# B&R Automation Studio project Embraco_LinkaNaOdlievanieRotorov_DokoncovaciaStanica_Rev2 (part 3)

#### Main.st - Init, cyclic, exit code
```iecst
PROGRAM _INIT
	(* Insert code here *)

END_PROGRAM

PROGRAM _CYCLIC

	//Volanie podprogramov//
	OvladanieGripra;
	OvladaniePojazdu;
	OvladanieZdvihu;

	//Volanie funkcie SequenceControl//
	SequenceControl(SC:= SC_VstupnyManipulator);

	//Reset sekcie //
	IF VstupManipulator_Reset OR NOT BezpOkruhOplotenia_Aktivovany OR PoruchaVstupManipulator THEN
		SC_VstupnyManipulator.Step:= 0;
	END_IF

	CASE SC_VstupnyManipulator.Step OF

		0:
			SC_VstupnyManipulator.StepName:='0 - Nulovanie';
			SC_OvlGripra.Step:= 0;
			SC_OvlServoPojazdu.Step:= 0;
			SC_OvlZdvihu.Step:= 0;
			VstupManipulator_Automat:= FALSE;
			VstupManipulator_KoniecVyroby:= FALSE;
			VstupManipulator_KoniecCyklu:= FALSE;
			VstupManipulator_Manual:= FALSE;
			VstupManipulator_PoINIT:= FALSE;
			VstupManipulator_Reset:= FALSE;
			VstupManipulator_PojazdVPOZICI:= FALSE;
			VstupManipulator_UkoncilCyklus:= FALSE;
			Zariadenie_PAUZA:= FALSE;
			VstupManipulator_OdobralRotor:= FALSE;
			IF BezpOkruhOplotenia_Aktivovany AND NOT PoruchaVstupManipulator THEN
				SC_VstupnyManipulator.ResetStep:= TRUE;
				SC_VstupnyManipulator.Step:= 1;
			END_IF

		1:
			SC_VstupnyManipulator.StepName:='1 - Rozhodnutie o cinnosti';
			IF VstupManipulator_Automat THEN
				SC_VstupnyManipulator.Step:= 2;
			ELSIF VstupManipulator_Manual THEN
				SC_VstupnyManipulator.Step:= 700;
			END_IF

		//********************************************************Inicializácia****************************************************************************//

		2:
			SC_VstupnyManipulator.StepName:='2 - Inicializacia - cakanie na spustenie';
			SC_VstupnyManipulator.IdleTime.PT:= T#500ms;
			SC_VstupnyManipulator.AlarmTime.PT:= T#5s;
			SC_VstupnyManipulator.IdleTime.IN:= TRUE;

			IF SC_VstupnyManipulator.IdleTime.Q THEN
				SC_VstupnyManipulator.ResetStep:= TRUE;
				SC_VstupnyManipulator.Step:= 3;
			END_IF

		3:
			SC_VstupnyManipulator.StepName:='3 - Inicializacia - kontrola home serva';
			SC_VstupnyManipulator.IdleTime.PT:= T#500ms;
			SC_VstupnyManipulator.AlarmTime.PT:= T#5s;

			IF Motion[1].status.DriveStatus.HomingOk THEN
				SC_VstupnyManipulator.ResetStep:= TRUE;
				SC_VstupnyManipulator.Step:= 5;
			ELSE
				SC_VstupnyManipulator.ResetStep:= TRUE;
				SC_VstupnyManipulator.Step:= 4;
			END_IF

		4:
			SC_VstupnyManipulator.StepName:='4 - Inicializacia - homing serva';
			SC_VstupnyManipulator.IdleTime.PT:= T#1s;
			SC_VstupnyManipulator.AlarmTime.PT:= T#5s;

			IF NOT SC_VstupnyManipulator.Switch1 THEN
				VstupManipulator_PojazdHOME:= TRUE;
				SC_VstupnyManipulator.Switch1:= TRUE;
			END_IF

			IF Motion[1].status.DriveStatus.HomingOk THEN
				SC_VstupnyManipulator.IdleTime.IN:= TRUE;
			END_IF

			IF Motion[1].status.DriveStatus.HomingOk AND SC_VstupnyManipulator.IdleTime.Q AND Motion[1].state.StandStill THEN
				SC_VstupnyManipulator.ResetStep:= TRUE;
				SC_VstupnyManipulator.Step:= 6;
			END_IF

		5:
			SC_VstupnyManipulator.StepName:='5 - Inicializacia - zodvihnutie gripra';
			SC_VstupnyManipulator.IdleTime.PT:= T#500ms;
			SC_VstupnyManipulator.AlarmTime.PT:= T#5s;

			IF NOT SC_VstupnyManipulator.Switch1 THEN
				Zdvih_Manipulatora:= TRUE;
				SC_VstupnyManipulator.Switch1:= TRUE;
			END_IF

			IF diVstupManipul_ZasunutyHore THEN
				SC_VstupnyManipulator.ResetStep:= TRUE;
				SC_VstupnyManipulator.Step:= 6;
			END_IF

		6:
			SC_VstupnyManipulator.StepName:='6 - Inicializacia - rozhodnutie o presunu manipulatora';
			SC_VstupnyManipulator.IdleTime.PT:= T#200ms;
			SC_VstupnyManipulator.AlarmTime.PT:= T#5s;

			IF diVstupManipul_GriperOtvoreny AND diVstupManipul_GriperZatvoreny THEN
				Alarmy[21]:= TRUE;
				PoruchaVstupManipulator:= TRUE;
			ELSIF diVstupManipul_GriperOtvoreny AND NOT diVstupManipul_GriperZatvoreny THEN
				VstupManipulator_PoINIT:= TRUE;
				SC_VstupnyManipulator.ResetStep:= TRUE;
				SC_VstupnyManipulator.Step:= 125;
			ELSIF NOT diVstupManipul_GriperOtvoreny AND diVstupManipul_GriperZatvoreny THEN
				VstupManipulator_PoINIT:= TRUE;
				SC_VstupnyManipulator.ResetStep:= TRUE;
				SC_VstupnyManipulator.Step:= 110;
			END_IF

		//********************************************************Automatický režim****************************************************************************//
		100:
			SC_VstupnyManipulator.StepName:='100 - Automaticky rezim - cakanie na odobratie rotora';
			SC_VstupnyManipulator.IdleTime.PT:= T#3s;
			SC_VstupnyManipulator.AlarmTime.PT:= T#5s;
			SC_VstupnyManipulator.IdleTime.IN:= TRUE;

			IF VstupManipulator_KoniecCyklu THEN
				SC_VstupnyManipulator.ResetStep:= TRUE;
				SC_VstupnyManipulator.Step:= 0;
			ELSIF diVstupManipul_GriperOtvoreny AND NOT diVstupManipul_GriperZatvoreny AND diVstupDopr_PritomnostRotora AND diVstupDopr_ZdvihRotora_HORE AND NOT VstupManipulator_KoniecVyroby THEN
				SC_VstupnyManipulator.ResetStep:= TRUE;
				SC_VstupnyManipulator.Step:= 101;
			ELSIF diVstupManipul_GriperZatvoreny AND NOT diVstupManipul_GriperOtvoreny THEN
				SC_VstupnyManipulator.ResetStep:= TRUE;
				SC_VstupnyManipulator.Step:= 108;
			ELSIF SC_VstupnyManipulator.IdleTime.Q AND Stol_Automat THEN
				VstupManipulator_UkoncilCyklus:= TRUE;
				SC_VstupnyManipulator.ResetStep:= TRUE;
				SC_VstupnyManipulator.Step:= 132;
			ELSIF VstupManipulator_KoniecVyroby AND NOT Stol_Automat THEN
				SC_VstupnyManipulator.ResetStep:= TRUE;
				SC_VstupnyManipulator.Step:= 0;
			END_IF

		101:
			SC_VstupnyManipulator.StepName:='101 - Automaticky rezim - zostup manipulatora nad vstupny dopravnik';
			SC_VstupnyManipulator.IdleTime.PT:= T#1s;
			SC_VstupnyManipulator.AlarmTime.PT:= T#5s;
			SC_VstupnyManipulator.IdleTime.IN:= TRUE;

			IF NOT SC_VstupnyManipulator.Switch1 THEN
				Zostup_Manipulatora:= TRUE;
				SC_VstupnyManipulator.Switch1:= TRUE;
			END_IF

			IF diVstupManipul_VysunutyDole THEN
				SC_VstupnyManipulator.ResetStep:= TRUE;
				SC_VstupnyManipulator.Step:= 102;
			END_IF

		102:
			SC_VstupnyManipulator.StepName:='102 - Automaticky rezim - zatvorenie gripra manipulatora';
			SC_VstupnyManipulator.IdleTime.PT:= T#500ms;
			SC_VstupnyManipulator.AlarmTime.PT:= T#5s;

			IF NOT SC_VstupnyManipulator.Switch1 THEN
				Zatvor_Griper:= TRUE;
				SC_VstupnyManipulator.Switch1:= TRUE;
			END_IF

			IF diVstupManipul_GriperZatvoreny THEN
				SC_VstupnyManipulator.ResetStep:= TRUE;
				SC_VstupnyManipulator.Step:= 103;
			END_IF

		103:
			SC_VstupnyManipulator.StepName:='103 - Automaticky rezim - otvorenie gripra manipulatora';
			SC_VstupnyManipulator.IdleTime.PT:= T#500ms;
			SC_VstupnyManipulator.AlarmTime.PT:= T#5s;

			IF NOT SC_VstupnyManipulator.Switch1 AND SC_OvlGripra.Step = 1 THEN
				Otvor_Griper:= TRUE;
				SC_VstupnyManipulator.Switch1:= TRUE;
			END_IF

			IF diVstupManipul_GriperOtvoreny THEN
				SC_VstupnyManipulator.ResetStep:= TRUE;
				SC_VstupnyManipulator.Step:= 104;
			END_IF

		104:
			SC_VstupnyManipulator.StepName:='104 - Automaticky rezim - zatvorenie gripra manipulatora';
			SC_VstupnyManipulator.IdleTime.PT:= T#500ms;
			SC_VstupnyManipulator.AlarmTime.PT:= T#5s;

			IF NOT SC_VstupnyManipulator.Switch1 AND SC_OvlGripra.Step = 1 THEN
				Zatvor_Griper:= TRUE;
				SC_VstupnyManipulator.Switch1:= TRUE;
			END_IF

			IF diVstupManipul_GriperZatvoreny THEN
				SC_VstupnyManipulator.ResetStep:= TRUE;
				SC_VstupnyManipulator.Step:= 108;
			END_IF

		108:
			SC_VstupnyManipulator.StepName:='102 - Automaticky rezim - zdvih manipulatora nad vstupny dopravnik, zistovanie NG kusu';
			SC_VstupnyManipulator.IdleTime.PT:= T#500ms;
			SC_VstupnyManipulator.AlarmTime.PT:= T#5s;
			SC_VstupnyManipulator.IdleTime.IN:= TRUE;

			IF NOT SC_VstupnyManipulator.Switch1 THEN
				Zdvih_Manipulatora:= TRUE;
				SC_VstupnyManipulator.Switch1:= TRUE;
			END_IF

			IF EDGEPOS(diVstupManipul_SpodSnimacNG_Kusu = TRUE) THEN
				IF diVstupManipul_HornSnimacNG_Kusu THEN
					VstupManipulator_Drzi_NG_Kus:= FALSE;
				ELSIF Zariadenie_PrebiehaRevorkRezim THEN
					VstupManipulator_Drzi_NG_Kus:= FALSE;
				ELSE
					VstupManipulator_Drzi_NG_Kus:= TRUE;
				END_IF
			END_IF

			IF diVstupManipul_ZasunutyHore THEN
				SC_VstupnyManipulator.ResetStep:= TRUE;
				SC_VstupnyManipulator.Step:= 110;
			END_IF

		110:
			SC_VstupnyManipulator.StepName:='104 - Automaticky rezim - presun manipulatora na poziciu vkladania';
			SC_VstupnyManipulator.IdleTime.PT:= T#500ms;
			SC_VstupnyManipulator.AlarmTime.PT:= T#5s;

			VstupManipulator_ZadanaPozMM:= TP_VstupManip_PoziciaUkladania; //9 mm

			IF NOT SC_VstupnyManipulator.Switch1 AND SC_OvlServoPojazdu.Step = 1 THEN
				ServoPojazd_Polohuj:= TRUE;
				SC_VstupnyManipulator.Switch1:= TRUE;
			END_IF

			IF VstupManipulator_PojazdVPOZICI AND (VstupManipulator_AktualPozMM = TP_VstupManip_PoziciaUkladania) THEN
				VstupManipulator_PojazdVPOZICI:= FALSE;
				SC_VstupnyManipulator.ResetStep:= TRUE;
				SC_VstupnyManipulator.Step:= 120;
			END_IF

		120:
			SC_VstupnyManipulator.StepName:='120 - Automaticky rezim - kontrola stola';
			SC_VstupnyManipulator.IdleTime.PT:= T#500ms;
			SC_VstupnyManipulator.AlarmTime.PT:= T#5s;

			IF Stol_PoINIT AND NOT VstupManipulator_UkoncilCyklus AND diStol_SnimacPolohyStola AND NOT diStol_PritomnostRotoraVstup THEN
				SC_VstupnyManipulator.ResetStep:= TRUE;
				SC_VstupnyManipulator.Step:= 122;
			ELSIF Stol_PoINIT AND NOT VstupManipulator_UkoncilCyklus AND diStol_SnimacPolohyStola AND diStol_PritomnostRotoraVstup THEN
				VstupManipulator_UkoncilCyklus:= TRUE;
				SC_VstupnyManipulator.ResetStep:= TRUE;
				SC_VstupnyManipulator.Step:= 132;
			ELSIF VstupManipulator_KoniecCyklu THEN
				SC_VstupnyManipulator.ResetStep:= TRUE;
				SC_VstupnyManipulator.Step:= 0;
			END_IF

		122:
			SC_VstupnyManipulator.StepName:='122 - Automaticky rezim - polozenie rotora na stol';
			SC_VstupnyManipulator.IdleTime.PT:= T#200ms;
			SC_VstupnyManipulator.AlarmTime.PT:= T#5s;
			SC_VstupnyManipulator.AlarmTime.IN:= TRUE;

			IF NOT SC_VstupnyManipulator.Switch1 AND diStol_SnimacPolohyStola AND NOT diStol_PritomnostRotoraVstup AND Stol.IN.CentrovanieVysunute=1 THEN
				Zostup_Manipulatora:= TRUE;
				SC_VstupnyManipulator.Switch1:= TRUE;
			END_IF

			IF diVstupManipul_ZdvihStredPoloha THEN
				SC_VstupnyManipulator.IdleTime.IN:= TRUE;
			END_IF

			IF diVstupManipul_VysunutyDole OR SC_VstupnyManipulator.IdleTime.Q THEN
				SC_VstupnyManipulator.ResetStep:= TRUE;
				SC_VstupnyManipulator.Step:= 123;
			END_IF

			IF SC_VstupnyManipulator.AlarmTime.Q THEN
				Alarmy[23]:= TRUE;
				PoruchaVstupManipulator:= TRUE;
			END_IF

		123:
			SC_VstupnyManipulator.StepName:='123 - Automaticky rezim - otvorenie gripra manipulatora';
			SC_VstupnyManipulator.IdleTime.PT:= T#500ms;
			SC_VstupnyManipulator.AlarmTime.PT:= T#5s;

			IF NOT SC_VstupnyManipulator.Switch1 THEN
				Otvor_Griper:= TRUE;
				SC_VstupnyManipulator.Switch1:= TRUE;
			END_IF

			IF diVstupManipul_GriperOtvoreny AND diVstupManipul_VysunutyDole THEN
				IF VstupManipulator_Drzi_NG_Kus THEN
					Stol_NG_KusNaStole:= TRUE;
				ELSE
					Stol_NG_KusNaStole:= FALSE;
				END_IF
				VstupManipulator_Drzi_NG_Kus:= FALSE;
				SC_VstupnyManipulator.ResetStep:= TRUE;
				SC_VstupnyManipulator.Step:= 124;
			END_IF

		124:
			SC_VstupnyManipulator.StepName:='124 - Automaticky rezim - zdvih manipulatora nad stol, vystavenie signalu ukoncenie cyklu';
			SC_VstupnyManipulator.IdleTime.PT:= T#500ms;
			SC_VstupnyManipulator.AlarmTime.PT:= T#5s;

			IF NOT SC_VstupnyManipulator.Switch1 AND SC_OvlZdvihu.Step = 1 THEN
				Zdvih_Manipulatora:= TRUE;
				Stol.OUT.CentrovanieVysunut:=0;
				Stol.OUT.CentrovanieZasunut:=1;
				SC_VstupnyManipulator.Switch1:= TRUE;
			END_IF

			IF diVstupManipul_ZasunutyHore AND Stol.IN.CentrovanieZasunute=1 THEN
				IF diStol_PritomnostRotoraVstup THEN
					VstupManipulator_UkoncilCyklus:= TRUE;
				END_IF
				SC_VstupnyManipulator.ResetStep:= TRUE;
				SC_VstupnyManipulator.Step:= 125;
			END_IF

		125:
			SC_VstupnyManipulator.StepName:='125 - Automaticky rezim - presun manipulatora na poziciu odoberania';
			SC_VstupnyManipulator.IdleTime.PT:= T#500ms;
			SC_VstupnyManipulator.AlarmTime.PT:= T#5s;

			VstupManipulator_ZadanaPozMM:= TP_VstupManip_PoziciaOdoberania;//602.0;

			IF NOT SC_VstupnyManipulator.Switch1 AND SC_OvlServoPojazdu.Step = 1 THEN
				ServoPojazd_Polohuj:= TRUE;
				SC_VstupnyManipulator.Switch1:= TRUE;
			END_IF

			IF VstupManipulator_PojazdVPOZICI AND (VstupManipulator_AktualPozMM = TP_VstupManip_PoziciaOdoberania) THEN
				VstupManipulator_PojazdVPOZICI:= FALSE;
				SC_VstupnyManipulator.ResetStep:= TRUE;
				SC_VstupnyManipulator.Step:= 100;
			END_IF

		132:
			SC_VstupnyManipulator.StepName:='132 - Automaticky rezim - cakanie na otocenie stola';
			SC_VstupnyManipulator.IdleTime.PT:= T#500ms;
			SC_VstupnyManipulator.AlarmTime.PT:= T#5s;

			IF NOT VstupManipulator_UkoncilCyklus THEN
				SC_VstupnyManipulator.ResetStep:= TRUE;
				SC_VstupnyManipulator.Step:= 100;
			ELSIF VstupManipulator_KoniecVyroby AND NOT Stol_Automat THEN
				SC_VstupnyManipulator.ResetStep:= TRUE;
				SC_VstupnyManipulator.Step:= 0;
			ELSIF VstupManipulator_KoniecCyklu THEN
				SC_VstupnyManipulator.ResetStep:= TRUE;
				SC_VstupnyManipulator.Step:= 0;
			END_IF

		//********************************************************Ručný režim***********************************************************************************//
		700:
			SC_VstupnyManipulator.StepName:='700 - Rucny rezim';

			//Polohovanie manipulátora//
			IF RR_PoziciaOdoberania AND SC_OvlServoPojazdu.Step = 1 THEN
				VstupManipul_Rychlost_MM_s:= TP_VstupManip_RychlostPojazdu;
				VstupManipulator_ZadanaPozMM:= TP_VstupManip_PoziciaOdoberania;
				ServoPojazd_Polohuj:= TRUE;
			ELSIF RR_PoziciaVkladaniaStol AND SC_OvlServoPojazdu.Step = 1 THEN
				VstupManipul_Rychlost_MM_s:= TP_VstupManip_RychlostPojazdu;
				VstupManipulator_ZadanaPozMM:= TP_VstupManip_PoziciaUkladania;
				ServoPojazd_Polohuj:= TRUE;
			END_IF

	END_CASE

				END_PROGRAM

PROGRAM _EXIT
				(* Insert code here *)

				END_PROGRAM
```

#### Variables.var - Local variables
```iecst
VAR
	SC_OvlGripra : SequenceControlTyp;
	Otvor_Griper : BOOL;
	Zatvor_Griper : BOOL;
	SC_OvlZdvihu : SequenceControlTyp;
	Zdvih_Manipulatora : BOOL;
	Zostup_Manipulatora : BOOL;
	SC_OvlServoPojazdu : SequenceControlTyp;
	ServoPojazd_JoggVPRED : BOOL;
	ServoPojazd_JoggVZAD : BOOL;
	ServoPojazd_Polohuj : BOOL;
	KonstantaPojazd_MM : REAL;
	KonstantaPojazd_Servo : REAL;
	RR_PoziciaOdoberania : BOOL;
	RR_PoziciaVkladaniaStol : BOOL;
END_VAR
```

#### OvladanieGripra.st
```iecst
ACTION OvladanieGripra:

	//Volanie funkcie SequenceControl//
	SequenceControl(SC:= SC_OvlGripra);

	CASE SC_OvlGripra.Step OF

		0:
			SC_OvlGripra.StepName:= '0 - Nulovanie';
			Otvor_Griper:= FALSE;
			Zatvor_Griper:= FALSE;
			doVstupManipul_GriperOTVOR:= FALSE;
			doVstupManipul_GriperZATVOR:= FALSE;
			IF SC_VstupnyManipulator.Step <> 0 THEN
				SC_OvlGripra.ResetStep:= TRUE;
				SC_OvlGripra.Step:= 1;
			END_IF

		1:
			SC_OvlGripra.StepName:= '1 - Rozhodnutie o cinnosti';
			IF Otvor_Griper THEN
				SC_OvlGripra.Step:= 10;
			ELSIF Zatvor_Griper THEN
				SC_OvlGripra.Step:= 20;
			END_IF

		10:
			SC_OvlGripra.StepName:= '10 - Otvorenie gripra';
			SC_OvlGripra.IdleTime.PT:= T#3s;
			SC_OvlGripra.AlarmTime.PT:= T#3s;

			IF VstupManipulator_Manual THEN
				SC_OvlGripra.IdleTime.IN:= TRUE;
			ELSE
				SC_OvlGripra.AlarmTime.IN:= TRUE;
			END_IF

			IF NOT SC_OvlGripra.Switch1 THEN
				doVstupManipul_GriperOTVOR:= TRUE;
				SC_OvlGripra.Switch1:= TRUE;
			END_IF

			IF SC_OvlGripra.AlarmTime.Q THEN
				Alarmy[21]:= TRUE;
				PoruchaVstupManipulator:= TRUE;
			END_IF

			IF diVstupManipul_GriperOtvoreny OR SC_OvlGripra.IdleTime.Q THEN
				SC_OvlGripra.ResetStep:= TRUE;
				SC_OvlGripra.Step:= 0;
			END_IF

		20:
			SC_OvlGripra.StepName:= '20 - Zatvorenie gripra';
			SC_OvlGripra.IdleTime.PT:= T#3s;
			SC_OvlGripra.AlarmTime.PT:= T#3s;

			IF VstupManipulator_Manual THEN
				SC_OvlGripra.IdleTime.IN:= TRUE;
			ELSE
				SC_OvlGripra.AlarmTime.IN:= TRUE;
			END_IF

			IF NOT SC_OvlGripra.Switch1 THEN
				doVstupManipul_GriperZATVOR:= TRUE;
				SC_OvlGripra.Switch1:= TRUE;
			END_IF

			IF SC_OvlGripra.AlarmTime.Q THEN
				Alarmy[20]:= TRUE;
				PoruchaVstupManipulator:= TRUE;
			END_IF

			IF diVstupManipul_GriperZatvoreny OR SC_OvlGripra.IdleTime.Q THEN
				SC_OvlGripra.ResetStep:= TRUE;
				SC_OvlGripra.Step:= 0;
			END_IF

	END_CASE

END_ACTION
```

#### OvladanieZdvihu.st
```iecst
ACTION OvladanieZdvihu:

	//Volanie funkcie SequenceControl//
	SequenceControl(SC:= SC_OvlZdvihu);

	CASE SC_OvlZdvihu.Step OF

		0:
			SC_OvlZdvihu.StepName:= '0 - Nulovanie';
			Zdvih_Manipulatora:= FALSE;
			Zostup_Manipulatora:= FALSE;
			doVstupManipul_ZDVIH:= FALSE;
			doVstupManipul_ZOSTUP:= FALSE;
			IF SC_VstupnyManipulator.Step <> 0 THEN
				SC_OvlZdvihu.ResetStep:= TRUE;
				SC_OvlZdvihu.Step:= 1;
			END_IF

		1:
			SC_OvlZdvihu.StepName:= '1 - Rozhodnutie o cinnosti';
			IF Zdvih_Manipulatora THEN
				SC_OvlZdvihu.Step:= 10;
			ELSIF Zostup_Manipulatora THEN
				SC_OvlZdvihu.Step:= 20;
			END_IF

		10:
			SC_OvlZdvihu.StepName:= '10 - Zdvih manipulatora';
			SC_OvlZdvihu.IdleTime.PT:= T#3s;
			SC_OvlZdvihu.AlarmTime.PT:= T#3s;

			IF VstupManipulator_Manual THEN
				SC_OvlZdvihu.IdleTime.IN:= TRUE;
			ELSE
				SC_OvlZdvihu.AlarmTime.IN:= TRUE;
			END_IF

			IF NOT SC_OvlZdvihu.Switch1 THEN
				doVstupManipul_ZDVIH:= TRUE;
				SC_OvlZdvihu.Switch1:= TRUE;
			END_IF

			IF SC_OvlZdvihu.AlarmTime.Q THEN
				Alarmy[22]:= TRUE;
				PoruchaVstupManipulator:= TRUE;
			END_IF

			IF diVstupManipul_ZasunutyHore OR SC_OvlZdvihu.IdleTime.Q THEN
				SC_OvlZdvihu.ResetStep:= TRUE;
				SC_OvlZdvihu.Step:= 0;
			END_IF

		20:
			SC_OvlZdvihu.StepName:= '20 - Zostup manipulatora';
			SC_OvlZdvihu.IdleTime.PT:= T#2s;
			SC_OvlZdvihu.AlarmTime.PT:= T#3s;
			SC_OvlZdvihu.IdleTime.IN:= TRUE;

			IF VstupManipulator_Manual THEN
				SC_OvlZdvihu.IdleTime.IN:= TRUE;
			ELSE
				SC_OvlZdvihu.AlarmTime.IN:= TRUE;
			END_IF

			IF NOT SC_OvlZdvihu.Switch1 THEN
				doVstupManipul_ZOSTUP:= TRUE;
				SC_OvlZdvihu.Switch1:= TRUE;
			END_IF

			IF EDGEPOS (diVstupManipul_ZdvihStredPoloha = TRUE) THEN
				doVstupManipul_ZDVIH:= TRUE;
			END_IF

			IF SC_OvlZdvihu.AlarmTime.Q THEN
				Alarmy[23]:= TRUE;
				PoruchaVstupManipulator:= TRUE;
			END_IF

			IF diVstupManipul_VysunutyDole OR SC_OvlZdvihu.IdleTime.Q THEN
				SC_OvlZdvihu.ResetStep:= TRUE;
				SC_OvlZdvihu.Step:= 0;
			END_IF

	END_CASE

END_ACTION
```

#### OvladaniePojazdu.st
```iecst
ACTION OvladaniePojazdu:

	//Prepočet rýchlosti pojazdu manipulátora//
	KonstantaPojazd_MM:= 8;  //8mm
	KonstantaPojazd_Servo:= 800; //počet jednotiek za 8mm

	VstupManipul_Rychlost_MM_s:= TP_VstupManip_RychlostPojazdu;
	VstupManipulator_RychlostPolohov:= (VstupManipul_Rychlost_MM_s / KonstantaPojazd_MM) * KonstantaPojazd_Servo;
	VstupManipulator_RychlJoggingu:= (VstupManipul_RychlostJog_MM_s / KonstantaPojazd_MM) * KonstantaPojazd_Servo;
	VstupManipulator_AktualPozMM;

	//Volanie funkcie SequenceControl//
	SequenceControl(SC:= SC_OvlServoPojazdu);

	CASE SC_OvlServoPojazdu.Step OF

		0:
			SC_OvlServoPojazdu.StepName:= '0 - Nulovanie';
			ServoPojazd_JoggVPRED:= FALSE;
			ServoPojazd_JoggVZAD:= FALSE;
			ServoPojazd_Polohuj:= FALSE;
			VstupManipulator_PojazdHOME:= FALSE;
			Motion[1].cmd.home:= FALSE;
			Motion[1].cmd.moveAbsolute:= FALSE;
			Motion[1].cmd.moveJogNeg:= FALSE;
			Motion[1].cmd.moveJogPos:= FALSE;
			VstupManipulator_PrebiehaHoming:= FALSE;
			IF NOT SC_OvlServoPojazdu.Switch1 AND Motion[1].status.DriveStatus.HomingOk THEN
				Motion[1].cmd.halt:= TRUE;
				SC_OvlServoPojazdu.Switch1:= TRUE;
			END_IF
			IF SC_VstupnyManipulator.Step <> 0 THEN
				SC_OvlServoPojazdu.ResetStep:= TRUE;
				SC_OvlServoPojazdu.Step:= 1;
			END_IF

		1:
			SC_OvlServoPojazdu.StepName:= '1 - Rozhodnutie o cinnosti';
			IF ServoPojazd_JoggVPRED THEN
				SC_OvlServoPojazdu.Step:= 10;
			ELSIF ServoPojazd_JoggVZAD THEN
				SC_OvlServoPojazdu.Step:= 20;
			ELSIF ServoPojazd_Polohuj THEN
				SC_OvlServoPojazdu.Step:= 30;
			ELSIF VstupManipulator_PojazdHOME THEN
				SC_OvlServoPojazdu.Step:= 40;
			END_IF

		10:
			SC_OvlServoPojazdu.StepName:= '10 - Jogging VPRED';
			SC_OvlServoPojazdu.IdleTime.PT:= T#3s;
			SC_OvlServoPojazdu.AlarmTime.PT:= T#3s;

			Motion[1].par.velocityJog:= VstupManipulator_RychlJoggingu;
			Motion[1].par.acc := (VstupManipulator_RychlJoggingu*10);
			Motion[1].par.dec := (VstupManipulator_RychlJoggingu*10);

			IF NOT SC_OvlServoPojazdu.Switch1 THEN
				Motion[1].cmd.moveJogPos:= TRUE;
				SC_OvlServoPojazdu.Switch1:= TRUE;
			END_IF

			IF NOT ServoPojazd_JoggVPRED OR diVstupManipul_PrednyLimitSnimac OR VstupManipulator_AktualPozMM >= 610 OR NOT diVstupManipul_ZasunutyHore THEN
				SC_OvlServoPojazdu.ResetStep:= TRUE;
				SC_OvlServoPojazdu.Step:= 0;
			END_IF

		20:
			SC_OvlServoPojazdu.StepName:= '10 - Jogging VZAD';
			SC_OvlServoPojazdu.IdleTime.PT:= T#3s;
			SC_OvlServoPojazdu.AlarmTime.PT:= T#3s;

			Motion[1].par.velocityJog:= VstupManipulator_RychlJoggingu;
			Motion[1].par.acc := (VstupManipulator_RychlJoggingu*10);
			Motion[1].par.dec := (VstupManipulator_RychlJoggingu*10);

			IF NOT SC_OvlServoPojazdu.Switch1 THEN
				Motion[1].cmd.moveJogNeg:= TRUE;
				SC_OvlServoPojazdu.Switch1:= TRUE;
			END_IF

			IF NOT ServoPojazd_JoggVZAD OR diVstupManipul_ZadnyLimitSnimac OR VstupManipulator_AktualPozMM < 0 OR NOT diVstupManipul_ZasunutyHore THEN
				SC_OvlServoPojazdu.ResetStep:= TRUE;
				SC_OvlServoPojazdu.Step:= 0;
			END_IF

		30:
			SC_OvlServoPojazdu.StepName:= '30 - Start polohovanie pojazdu';
			SC_OvlServoPojazdu.IdleTime.PT:= T#100ms;
			SC_OvlServoPojazdu.AlarmTime.PT:= T#3s;
			SC_OvlServoPojazdu.IdleTime.IN:= TRUE;

			Motion[1].par.velocity:= VstupManipulator_RychlostPolohov;
			Motion[1].par.acc := (VstupManipulator_RychlostPolohov*10);
			Motion[1].par.dec := (VstupManipulator_RychlostPolohov*10);
			Motion[1].par.position:= (VstupManipulator_ZadanaPozMM * 100);

			IF NOT SC_OvlServoPojazdu.Switch1 AND SC_OvlServoPojazdu.IdleTime.Q THEN
				Motion[1].cmd.moveAbsolute:= TRUE;
				SC_OvlServoPojazdu.Switch1:= TRUE;
			END_IF

			IF NOT Motion[1].state.StandStill THEN
				SC_OvlServoPojazdu.ResetStep:= TRUE;
				SC_OvlServoPojazdu.Step:= 31;
			ELSIF (VstupManipulator_AktualPozMM = VstupManipulator_ZadanaPozMM) THEN
				SC_OvlServoPojazdu.ResetStep:= TRUE;
				SC_OvlServoPojazdu.Step:= 31;
			END_IF

		31:

			SC_OvlServoPojazdu.StepName:= '31 - Ukoncenie polohovanie pojazdu';
			SC_OvlServoPojazdu.IdleTime.PT:= T#3s;
			SC_OvlServoPojazdu.AlarmTime.PT:= T#3s;

			IF Motion[1].state.StandStill AND (VstupManipulator_AktualPozMM = VstupManipulator_ZadanaPozMM) THEN
				VstupManipulator_PojazdVPOZICI:= TRUE;
				SC_OvlServoPojazdu.ResetStep:= TRUE;
				SC_OvlServoPojazdu.Step:= 0;
			END_IF

			IF diVstupManipul_PrednyLimitSnimac OR diVstupManipul_ZadnyLimitSnimac THEN
				Alarmy[26]:= TRUE;
				PoruchaVstupManipulator:= TRUE;
			END_IF

		40:
			SC_OvlServoPojazdu.StepName:= '40 - Homing,zdvihnutie gripra';
			SC_OvlServoPojazdu.IdleTime.PT:= T#3s;
			SC_OvlServoPojazdu.AlarmTime.PT:= T#3s;

			IF NOT SC_OvlServoPojazdu.Switch1 THEN
				VstupManipulator_PrebiehaHoming:= TRUE;
				Zdvih_Manipulatora:= TRUE;
				SC_OvlServoPojazdu.Switch1:= TRUE;
			END_IF

			IF diVstupManipul_ZasunutyHore THEN
				SC_OvlServoPojazdu.ResetStep:= TRUE;
				SC_OvlServoPojazdu.Step:= 41;
			END_IF

		41:
			SC_OvlServoPojazdu.StepName:= '41 - Homing,spustenie';
			SC_OvlServoPojazdu.IdleTime.PT:= T#3s;
			SC_OvlServoPojazdu.AlarmTime.PT:= T#3s;

			IF NOT SC_OvlServoPojazdu.Switch1 THEN
				Motion[1].cmd.home:= TRUE;
				SC_OvlServoPojazdu.Switch1:= TRUE;
			END_IF

			IF Motion[1].state.Homing THEN
				SC_OvlServoPojazdu.ResetStep:= TRUE;
				SC_OvlServoPojazdu.Step:= 42;
			END_IF

		42:
			SC_OvlServoPojazdu.StepName:= '42 - Homing,ukoncenie';
			SC_OvlServoPojazdu.IdleTime.PT:= T#3s;
			SC_OvlServoPojazdu.AlarmTime.PT:= T#3s;

			IF Motion[1].status.DriveStatus.HomingOk AND Motion[1].state.StandStill THEN
				SC_OvlServoPojazdu.ResetStep:= TRUE;
				SC_OvlServoPojazdu.Step:= 0;
			END_IF

	END_CASE

END_ACTION
```

### Program Logical/Program/OtocnyStol (IEC)

#### Main.st - Init, cyclic, exit code
```iecst
PROGRAM _INIT
	(* Insert code here *)

END_PROGRAM

PROGRAM _CYCLIC

	//Volanie podprogramov//
    OvladanieOtacania;

    //Volanie funkcie SequenceControl//
    SequenceControl(SC:= SC_Stol);

    //Blokovanie otáčania stola//
    IF diMeranie_ZdvihSpodnaPoloha AND
        diRazenie_ZdvihSpodnaPoloha AND
        Vyrazanie.IN.VyrazanieJeDole AND
        diValcovanie_ZdvihSpodnaPoloha AND
        (diVstupManipul_ZasunutyHore OR VstupManipulator_AktualPozMM > 15) AND
        (diVystupManipul_ZasunutyHore OR VystupManipulator_AktualPozMM > 15) AND
        NOT diValcovanie_PritomnostNastroja AND
        diValc2_ZdvihRotoraZasunuty AND
        Vyrazanie.IN.CentrovanieOtvorene THEN
        Stol_BlokovanieOtacania:= FALSE;
    ELSE
        Stol_BlokovanieOtacania:= TRUE;
    END_IF

    //Reset sekcie //
    IF Stol_Reset OR NOT BezpOkruhOplotenia_Aktivovany OR PoruchaOtocnyStol THEN
        SC_Stol.Step:= 0;
    END_IF

    CASE SC_Stol.Step OF

        0:
            SC_Stol.StepName:='0 - Nulovanie';
            SC_OvlStola.Step:= 0;
            Stol_Automat:= FALSE;
            Stol_KoniecVyroby:= FALSE;
            Stol_KoniecCyklu:= FALSE;
            Stol_Manual:= FALSE;
            Stol_PoINIT:= FALSE;
            Stol_Reset:= FALSE;
            Stol_PrebehloOtocenie:= FALSE;
            Stol_CakaNaVstupnyManipulator:= FALSE;
            Stol_CakaNaStrihanie:= FALSE;
            Stol_CakaNaRazenie:= FALSE;
            Stol_CakaNaValcovanie:= FALSE;
            Stol_CakaNaMeranie:= FALSE;
            Stol_CakaNaVystupnyManipulator:= FALSE;
            //			Stol_Pozicia_1:= 0;
            //			Stol_Pozicia_2:= 0;
            //			Stol_Pozicia_3:= 0;
            PocetOtoceniStola:= 0;
            Stol_StavPrazdnyStol:= FALSE;
            CasTaktTime2.IN:= FALSE;
            CasTaktTime1.IN:= FALSE;
            TP_Stol_Centrovanie_VYSUN:= FALSE;
            TP_Stol_Centrovanie_ZASUN:= FALSE;
            IF BezpOkruhOplotenia_Aktivovany AND NOT PoruchaOtocnyStol THEN
                SC_Stol.ResetStep:= TRUE;
                SC_Stol.Step:= 1;
            END_IF

        1:
            SC_Stol.StepName:='1 - Rozhodnutie o cinnosti';
            IF Stol_Automat THEN
                CisloChyby:= 0;
                SC_Stol.Step:= 2;
            ELSIF Stol_Manual THEN
                SC_Stol.Step:= 700;
            END_IF

            //********************************************************Inicializácia****************************************************************************//

        2:
            SC_Stol.StepName:='2 - Inicializacia - cakanie na spustenie';
            SC_Stol.IdleTime.PT:= T#500ms;
            SC_Stol.AlarmTime.PT:= T#5s;
            SC_Stol.IdleTime.IN:= TRUE;

            IF SC_Stol.IdleTime.Q THEN
                SC_Stol.ResetStep:= TRUE;
                SC_Stol.Step:= 3;
            END_IF

        3:
            SC_Stol.StepName:='2 - Inicializacia - rozhodnutie o otoceni stola';
            SC_Stol.IdleTime.PT:= T#500ms;
            SC_Stol.AlarmTime.PT:= T#5s;

            IF diStol_SnimacPolohyStola THEN
                Stol.OUT.CentrovanieVysunut:=1;
                Stol.OUT.CentrovanieZasunut:=0;
                Stol_PoINIT:= TRUE;
                SC_Stol.ResetStep:= TRUE;
                IF Stol.IN.CentrovanieVysunute=1 THEN
                    SC_Stol.Step:= 100;
                END_IF
            ELSE
                SC_Stol.ResetStep:= TRUE;
                SC_Stol.Step:= 4;
            END_IF

        4:
            SC_Stol.StepName:='4 - Inicializacia - otocenie stola vpred';
            SC_Stol.IdleTime.PT:= T#500ms;
            SC_Stol.AlarmTime.PT:= T#5s;

            IF NOT SC_Stol.Switch1 AND NOT Stol_BlokovanieOtacania THEN
                Otacaj_VPRED:= TRUE;
                SC_Stol.Switch1:= TRUE;
            END_IF

            IF diStol_SnimacPolohyStola AND Stol_PrebehloOtocenie THEN
                Stol_PrebehloOtocenie:= FALSE;
                Stol_PoINIT:= TRUE;
                SC_Stol.ResetStep:= TRUE;
                SC_Stol.Step:= 100;
            END_IF

            //********************************************************Automatický režim****************************************************************************//
        100:
            SC_Stol.StepName:='100 - Automaticky rezim - cakanie na ukoncenie cyklov jednotlivych pracovisk';
            SC_Stol.IdleTime.PT:= T#500ms;
            SC_Stol.AlarmTime.PT:= T#5s;

            IF VstupManipulator_UkoncilCyklus AND Strihanie_UkoncilCyklus AND Razenie_UkoncilCyklus AND Valcovanie_UkoncilCyklus AND Valcovanie2_UkoncilCyklus AND Meranie_UkoncilCyklus AND VystupManipulator_UkoncilCyklus AND NOT Stol_NG_KusNaStole THEN
                IF NOT CasTaktTime1.IN AND NOT CasTaktTime2.IN THEN
                    CasTaktTime1.IN:= TRUE;
                ELSIF CasTaktTime1.IN AND NOT CasTaktTime2.IN THEN
                    Zariadenie_TaktTime:= TIME_TO_REAL(CasTaktTime1.ET);
                    TP_Zariadenie_TaktTime:= (Zariadenie_TaktTime / 1000);
                    CasTaktTime2.IN:= TRUE;
                    CasTaktTime1.IN:= FALSE;
                ELSIF NOT CasTaktTime1.IN AND CasTaktTime2.IN THEN
                    Zariadenie_TaktTime:= TIME_TO_REAL(CasTaktTime2.ET);
                    TP_Zariadenie_TaktTime:= (Zariadenie_TaktTime / 1000);
                    CasTaktTime1.IN:= TRUE;
                    CasTaktTime2.IN:= FALSE;
                END_IF
                SC_Stol.ResetStep:= TRUE;
                SC_Stol.Step:= 101;
            ELSIF VstupManipulator_UkoncilCyklus AND Strihanie_UkoncilCyklus AND Razenie_UkoncilCyklus AND Valcovanie_UkoncilCyklus AND Valcovanie2_UkoncilCyklus AND Meranie_UkoncilCyklus AND VystupManipulator_UkoncilCyklus AND Stol_NG_KusNaStole THEN
                Stol_NG_KusNaStole:= FALSE;
                SC_Stol.ResetStep:= TRUE;
                SC_Stol.Step:= 105;
            ELSIF Stol_KoniecCyklu AND NOT VstupManipulator_Automat AND NOT Strihanie_Automat AND NOT Razenie_Automat AND NOT Valcovanie_Automat AND NOT Valcovanie2_Automat AND NOT Meranie_Automat AND NOT VystupManipulator_Automat THEN
                SC_Stol.ResetStep:= TRUE;
                SC_Stol.Step:= 0;
            END_IF

        101:
            SC_Stol.StepName:='101 - Automaticky rezim - otocenie stola vpred,prepisanie bufferov ';
            SC_Stol.IdleTime.PT:= T#500ms;
            SC_Stol.AlarmTime.PT:= T#5s;

            IF NOT SC_Stol.Switch2 THEN
                IF NOT diStol_PritomnostRotoraVstup AND NOT diStol_PritomnostRotoraVystup AND 	NOT Vyrazanie.IN.KusPritomny AND NOT diRazenie_PritomnostRotora AND NOT diValcovanie_PritomnostRotora AND NOT diValc2_PritomnostRotora AND NOT diMeranie_PritomnostRotora THEN
                    PocetOtoceniStola:= PocetOtoceniStola + 1;
                ELSE
                    PocetOtoceniStola:= 0;
                END_IF
                IF PocetOtoceniStola > 3 THEN
                    Stol_StavPrazdnyStol:= TRUE;
                ELSE
                    Stol_StavPrazdnyStol:= FALSE;
                END_IF
                SC_Stol.Switch2:= TRUE;
            END_IF

            IF NOT SC_Stol.Switch1 AND NOT Stol_BlokovanieOtacania AND diStol_NaliatokOdstrihnuty THEN
                Otacaj_VPRED:= TRUE;
                SC_Stol.Switch1:= TRUE;
            END_IF

            IF NOT diStol_NaliatokOdstrihnuty THEN
                SC_Stol.AlarmTime.IN:= TRUE;
            ELSIF Stol_BlokovanieOtacania THEN
                SC_Stol.AlarmTime.IN:= TRUE;
            ELSE
                SC_Stol.AlarmTime.IN:= FALSE;
            END_IF

            IF SC_Stol.AlarmTime.Q THEN
                IF NOT diStol_NaliatokOdstrihnuty THEN
                    Alarmy[34]:= TRUE;
                END_IF
                IF Stol_BlokovanieOtacania THEN
                    IF NOT diMeranie_ZdvihSpodnaPoloha THEN
                        CisloChyby:= 1;
                    ELSIF NOT diRazenie_ZdvihSpodnaPoloha THEN
                        CisloChyby:= 2;
                    ELSIF NOT Vyrazanie.IN.VyrazanieJeDole THEN
                        CisloChyby:= 3;
                    ELSIF NOT diValcovanie_ZdvihSpodnaPoloha THEN
                        CisloChyby:= 4;
                    ELSIF diValcovanie_PritomnostNastroja THEN
                        CisloChyby:= 5;
                    ELSIF NOT Vyrazanie.IN.CentrovanieOtvorene THEN
                        CisloChyby:= 6;
                    ELSIF (NOT diVstupManipul_ZasunutyHore AND VstupManipulator_AktualPozMM < 15) THEN
                        CisloChyby:= 7;
                    ELSIF (NOT diVystupManipul_ZasunutyHore AND VystupManipulator_AktualPozMM < 15) THEN
                        CisloChyby:= 8;
                    END_IF
                    Alarmy[33]:= TRUE;
                END_IF
                PoruchaOtocnyStol:= TRUE;
            END_IF

            IF diStol_SnimacPolohyStola AND Stol_PrebehloOtocenie THEN
                Stol_PrebehloOtocenie:= FALSE;
                Stol_Pozicia_3:= Stol_Pozicia_2;
                Stol_Pozicia_2:= Stol_Pozicia_1;
                Stol_Pozicia_1:= 0;
                SC_Stol.ResetStep:= TRUE;
                SC_Stol.Step:= 102;
            END_IF

        102:
            SC_Stol.StepName:='102 - Automaticky rezim - kontrola vyprazdnenia stola';
            SC_Stol.IdleTime.PT:= T#500ms;
            SC_Stol.AlarmTime.PT:= T#5s;

            IF NOT Stol_StavPrazdnyStol THEN
                Stol_PrebehloOtocenie:= FALSE;
                VstupManipulator_UkoncilCyklus:= FALSE;
                Strihanie_UkoncilCyklus:= FALSE;
                Razenie_UkoncilCyklus:= FALSE;
                Valcovanie_UkoncilCyklus:= FALSE;
                Valcovanie2_UkoncilCyklus:= FALSE;
                Meranie_UkoncilCyklus:= FALSE;
                VystupManipulator_UkoncilCyklus:= FALSE;
                SC_Stol.ResetStep:= TRUE;
                SC_Stol.Step:= 100;
            ELSIF NOT Stol_KoniecVyroby AND Stol_StavPrazdnyStol AND diVstupDopr_PritomnostRotora THEN
                Stol_PrebehloOtocenie:= FALSE;
                VstupManipulator_UkoncilCyklus:= FALSE;
                Strihanie_UkoncilCyklus:= FALSE;
                Razenie_UkoncilCyklus:= FALSE;
                Valcovanie_UkoncilCyklus:= FALSE;
                Valcovanie2_UkoncilCyklus:= FALSE;
                Meranie_UkoncilCyklus:= FALSE;
                VystupManipulator_UkoncilCyklus:= FALSE;
                SC_Stol.ResetStep:= TRUE;
                SC_Stol.Step:= 100;
            ELSIF Stol_KoniecVyroby AND NOT Stol_StavPrazdnyStol THEN
                Stol_PrebehloOtocenie:= FALSE;
                VstupManipulator_UkoncilCyklus:= FALSE;
                Strihanie_UkoncilCyklus:= FALSE;
                Razenie_UkoncilCyklus:= FALSE;
                Valcovanie_UkoncilCyklus:= FALSE;
                Valcovanie2_UkoncilCyklus:= FALSE;
                Meranie_UkoncilCyklus:= FALSE;
                VystupManipulator_UkoncilCyklus:= FALSE;
                SC_Stol.ResetStep:= TRUE;
                SC_Stol.Step:= 100;
            ELSIF Stol_KoniecVyroby AND Stol_StavPrazdnyStol THEN
                SC_Stol.ResetStep:= TRUE;
                SC_Stol.Step:= 0;
            ELSIF Stol_KoniecCyklu AND Stol_StavPrazdnyStol THEN
                SC_Stol.ResetStep:= TRUE;
                SC_Stol.Step:= 0;
            END_IF

            //Vyhodenie NG kusu//

        105:
            SC_Stol.StepName:='105 - Automaticky rezim - otocenie stola vzad';
            SC_Stol.IdleTime.PT:= T#500ms;
            SC_Stol.AlarmTime.PT:= T#5s;

            IF NOT SC_Stol.Switch1 AND NOT Stol_BlokovanieOtacania THEN
                Otacaj_VZAD:= TRUE;
                SC_Stol.Switch1:= TRUE;
            END_IF

            IF diStol_SnimacPolohyStola AND Stol_PrebehloOtocenie THEN
                VystupManipulator_OdoberNGKus:= TRUE;
                Stol_PrebehloOtocenie:= FALSE;
                SC_Stol.ResetStep:= TRUE;
                SC_Stol.Step:= 106;
            END_IF

        106:
            SC_Stol.StepName:='106 - Automaticky rezim - odobratie NG kusu';
            SC_Stol.IdleTime.PT:= T#500ms;
            SC_Stol.AlarmTime.PT:= T#5s;

            VystupManipulator_UkoncilCyklus:= FALSE;
            SC_Stol.ResetStep:= TRUE;
            SC_Stol.Step:= 107;

        107:
            SC_Stol.StepName:='107 - Automaticky rezim - ukoncenie odobratie NG kusu';
            SC_Stol.IdleTime.PT:= T#500ms;
            SC_Stol.AlarmTime.PT:= T#5s;

            IF VystupManipulator_UkoncilCyklus AND NOT diStol_PritomnostRotoraVystup THEN
                SC_Stol.ResetStep:= TRUE;
                SC_Stol.Step:= 108;
            END_IF

        108:
            SC_Stol.StepName:='108 - Automaticky rezim - otocenie stola vpred';
            SC_Stol.IdleTime.PT:= T#500ms;
            SC_Stol.AlarmTime.PT:= T#5s;

            IF NOT SC_Stol.Switch1 AND NOT Stol_BlokovanieOtacania AND diStol_NaliatokOdstrihnuty THEN
                Otacaj_VPRED:= TRUE;
                SC_Stol.Switch1:= TRUE;
            END_IF

            IF diStol_SnimacPolohyStola AND Stol_PrebehloOtocenie THEN
                Stol_PrebehloOtocenie:= FALSE;
                SC_Stol.ResetStep:= TRUE;
                SC_Stol.Step:= 109;
            END_IF

            IF NOT diStol_NaliatokOdstrihnuty THEN
                SC_Stol.AlarmTime.IN:= TRUE;
            ELSIF Stol_BlokovanieOtacania THEN
                SC_Stol.AlarmTime.IN:= TRUE;
            ELSE
                SC_Stol.AlarmTime.IN:= FALSE;
            END_IF

            IF SC_Stol.AlarmTime.Q THEN
                IF NOT diStol_NaliatokOdstrihnuty THEN
                    Alarmy[34]:= TRUE;
                END_IF
                IF Stol_BlokovanieOtacania THEN
                    IF NOT diMeranie_ZdvihSpodnaPoloha THEN
                        CisloChyby:= 1;
                    ELSIF NOT diRazenie_ZdvihSpodnaPoloha THEN
                        CisloChyby:= 2;
                    ELSIF NOT Vyrazanie.IN.VyrazanieJeDole THEN
                        CisloChyby:= 3;
                    ELSIF NOT diValcovanie_ZdvihSpodnaPoloha THEN
                        CisloChyby:= 4;
                    ELSIF diValcovanie_PritomnostNastroja THEN
                        CisloChyby:= 5;
                    ELSIF NOT Vyrazanie.IN.CentrovanieOtvorene THEN
                        CisloChyby:= 6;
                    ELSIF (NOT diVstupManipul_ZasunutyHore AND VstupManipulator_AktualPozMM < 15) THEN
                        CisloChyby:= 7;
                    ELSIF (NOT diVystupManipul_ZasunutyHore AND VystupManipulator_AktualPozMM < 15) THEN
                        CisloChyby:= 8;
                    END_IF
                    Alarmy[33]:= TRUE;
                END_IF
                PoruchaOtocnyStol:= TRUE;
            END_IF

        109:
            SC_Stol.StepName:='109 - Automaticky rezim - vystavenie signalu pre vstupny manipulator';
            SC_Stol.IdleTime.PT:= T#500ms;
            SC_Stol.AlarmTime.PT:= T#5s;

            VstupManipulator_UkoncilCyklus:= FALSE;
            SC_Stol.ResetStep:= TRUE;
            SC_Stol.Step:= 110;

        110:
            SC_Stol.StepName:='110 - Automaticky rezim - cakanie na ukoncenie cyklu vstupneho manipulatora';
            SC_Stol.IdleTime.PT:= T#500ms;
            SC_Stol.AlarmTime.PT:= T#5s;

            IF VstupManipulator_UkoncilCyklus THEN
                SC_Stol.ResetStep:= TRUE;
                SC_Stol.Step:= 100;
            ELSIF Stol_KoniecCyklu THEN
                SC_Stol.ResetStep:= TRUE;
                SC_Stol.Step:= 0;
            END_IF

            //********************************************************Ručný režim***********************************************************************************//
        700:
            SC_Stol.StepName:='700 - Rucny rezim';

            //Ovládanie centrovania rotora na vstupe stola//
            IF TP_Stol_Centrovanie_VYSUN AND diStol_SnimacPolohyStola THEN
                Stol.OUT.CentrovanieVysunut:=1;
                Stol.OUT.CentrovanieZasunut:=0;
                TP_Stol_Centrovanie_VYSUN:= FALSE;
            ELSIF TP_Stol_Centrovanie_ZASUN THEN
                Stol.OUT.CentrovanieVysunut:=0;
                Stol.OUT.CentrovanieZasunut:=1;
                TP_Stol_Centrovanie_ZASUN:= FALSE;
            END_IF

            //Ovládanie otáčania stola//
            IF Stol_RR_OtacajVPRED THEN
                IF NOT Stol_BlokovanieOtacania THEN
                    Otacaj_VPRED:= TRUE;
                END_IF
                Stol_RR_OtacajVPRED:= FALSE;
            ELSIF Stol_RR_OtacajVZAD THEN
                IF NOT Stol_BlokovanieOtacania THEN
                    Otacaj_VZAD:= TRUE;
                END_IF
                Stol_RR_OtacajVZAD:= FALSE;
            END_IF

    END_CASE

    CasTaktTime1.PT:= T#10m;
    CasTaktTime1();
    CasTaktTime2.PT:= T#10m;
    CasTaktTime2();

					END_PROGRAM

PROGRAM _EXIT
					(* Insert code here *)

					END_PROGRAM
```

#### Variables.var - Local variables
```iecst
VAR
	SC_OvlStola : SequenceControlTyp;
	Otacaj_VPRED : BOOL;
	Otacaj_VZAD : BOOL;
	PocetOtoceniStola : USINT;
	CasTaktTime1 : TON;
	CasTaktTime2 : TON;
	CisloChyby : USINT;
END_VAR
```

#### OvladanieOtacania.st
```iecst
ACTION OvladanieOtacania:

	//Volanie funkcie SequenceControl//
	SequenceControl(SC:= SC_OvlStola);

	CASE SC_OvlStola.Step OF

		0:
			SC_OvlStola.StepName:= '0 - Nulovanie';
			Otacaj_VPRED:= FALSE;
			Otacaj_VZAD:= FALSE;
			doStol_ODBRZDENIE:= FALSE;
			doStol_OtacajVPRED:= FALSE;
			doStol_OtacajVZAD:= FALSE;
			Stol.OUT.CentrovanieVysunut:=0;
			Stol.OUT.CentrovanieZasunut:=0;

			IF SC_Stol.Step <> 0 THEN
				SC_OvlStola.ResetStep:= TRUE;
				SC_OvlStola.Step:= 1;
			END_IF

		1:
			SC_OvlStola.StepName:= '1 - Rozhodnutie o cinnosti';
			IF Otacaj_VPRED THEN
				SC_OvlStola.Step:= 10;
			ELSIF Otacaj_VZAD THEN
				SC_OvlStola.Step:= 20;
			END_IF

		10:
			SC_OvlStola.StepName:= '10 - Zasunutie centrovania';
			SC_OvlStola.IdleTime.PT:= T#7s;
			SC_OvlStola.AlarmTime.PT:= T#7s;
			IF Stol_Manual THEN
				SC_OvlStola.IdleTime.IN:= TRUE;
			ELSE
				SC_OvlStola.AlarmTime.IN:= TRUE;
			END_IF

			IF NOT SC_OvlStola.Switch1 THEN
				Stol.OUT.CentrovanieVysunut:=0;
				Stol.OUT.CentrovanieZasunut:=1;
				SC_OvlStola.Switch1:= TRUE;
			END_IF

			IF Stol.IN.CentrovanieZasunute=1 THEN
				SC_OvlStola.ResetStep:= TRUE;
				SC_OvlStola.Step:= 11;
			END_IF

		11:
			SC_OvlStola.StepName:= '11 - Spustenie otacania stola vpred';
			SC_OvlStola.IdleTime.PT:= T#7s;
			SC_OvlStola.AlarmTime.PT:= T#7s;
			IF Stol_Manual THEN
				SC_OvlStola.IdleTime.IN:= TRUE;
			ELSE
				SC_OvlStola.AlarmTime.IN:= TRUE;
			END_IF

			IF NOT SC_OvlStola.Switch1 AND NOT Stol_BlokovanieOtacania THEN
				doStol_ODBRZDENIE:= TRUE;
				doStol_OtacajVPRED:= TRUE;
				SC_OvlStola.Switch1:= TRUE;
			END_IF

            IF doStol_OtacajVPRED AND NOT diStol_SnimacPolohyStola THEN
                SC_OvlStola.ResetStep:= TRUE;
				SC_OvlStola.Step:= 12;
			END_IF

		12:
			SC_OvlStola.StepName:= '12 - Zastavenie otacania stola vpred';
			SC_OvlStola.IdleTime.PT:= T#7s;
			SC_OvlStola.AlarmTime.PT:= T#7s;

			IF EDGEPOS (diStol_SnimacPolohyStola = TRUE) THEN
				//Stol_PrebehloOtocenie:= TRUE;
				doStol_ODBRZDENIE:= FALSE;
				doStol_OtacajVPRED:= FALSE;
				SC_OvlStola.ResetStep:= TRUE;
				SC_OvlStola.Step:= 13;
			ELSIF SC_OvlStola.IdleTime.Q THEN
				doStol_ODBRZDENIE:= FALSE;
				doStol_OtacajVPRED:= FALSE;
				SC_OvlStola.ResetStep:= TRUE;
				SC_OvlStola.Step:= 0;
			END_IF

            IF SC_OvlStola.AlarmTime.Q THEN
				Alarmy[31]:= TRUE;
				PoruchaOtocnyStol:= TRUE;
			END_IF

		13:
			SC_OvlStola.StepName:= '13 - Vysunutie centrovania';
			SC_OvlStola.IdleTime.PT:= T#7s;
			SC_OvlStola.AlarmTime.PT:= T#7s;
			IF Stol_Manual THEN
				SC_OvlStola.IdleTime.IN:= TRUE;
			ELSE
				SC_OvlStola.AlarmTime.IN:= TRUE;
			END_IF

			IF NOT SC_OvlStola.Switch1 THEN
				doStol_ODBRZDENIE:= FALSE;
				doStol_OtacajVPRED:= FALSE;
				Stol.OUT.CentrovanieVysunut:=1;
				Stol.OUT.CentrovanieZasunut:=0;
				SC_OvlStola.Switch1:= TRUE;
			END_IF

			IF Stol.IN.CentrovanieVysunute=1 THEN
				Stol_PrebehloOtocenie:= TRUE;
				SC_OvlStola.ResetStep:= TRUE;
				SC_OvlStola.Step:= 0;
			END_IF

		20:
			SC_OvlStola.StepName:= '20 - Zasunutie centrovania';
			SC_OvlStola.IdleTime.PT:= T#7s;
			SC_OvlStola.AlarmTime.PT:= T#7s;
			IF Stol_Manual THEN
				SC_OvlStola.IdleTime.IN:= TRUE;
			ELSE
				SC_OvlStola.AlarmTime.IN:= TRUE;
			END_IF

			IF NOT SC_OvlStola.Switch1 THEN
				Stol.OUT.CentrovanieVysunut:=0;
				Stol.OUT.CentrovanieZasunut:=1;
				SC_OvlStola.Switch1:= TRUE;
			END_IF

			IF Stol.IN.CentrovanieZasunute=1 THEN
				SC_OvlStola.ResetStep:= TRUE;
				SC_OvlStola.Step:= 21;
			END_IF

		21:
			SC_OvlStola.StepName:= '21 - Spustenie otacania stola vzad';
			SC_OvlStola.IdleTime.PT:= T#7s;
			SC_OvlStola.AlarmTime.PT:= T#7s;
			IF Stol_Manual THEN
				SC_OvlStola.IdleTime.IN:= TRUE;
			ELSE
				SC_OvlStola.AlarmTime.IN:= TRUE;
			END_IF

			Stol.OUT.CentrovanieVysunut:=0;
			Stol.OUT.CentrovanieZasunut:=1;

			IF NOT SC_OvlStola.Switch1 AND NOT Stol_BlokovanieOtacania THEN
				doStol_ODBRZDENIE:= TRUE;
				doStol_OtacajVZAD:= TRUE;
				SC_OvlStola.Switch1:= TRUE;
			END_IF

            IF doStol_OtacajVZAD AND NOT diStol_SnimacPolohyStola THEN
                SC_OvlStola.ResetStep:= TRUE;
				SC_OvlStola.Step:= 22;
			END_IF

		22:
			SC_OvlStola.StepName:= '22 - Zastavenie otacania stola vzad';
			SC_OvlStola.IdleTime.PT:= T#7s;
			SC_OvlStola.AlarmTime.PT:= T#7s;

			IF EDGEPOS (diStol_SnimacPolohyStola = TRUE) THEN
				//Stol_PrebehloOtocenie:= TRUE;
				doStol_ODBRZDENIE:= FALSE;
				doStol_OtacajVPRED:= FALSE;
				SC_OvlStola.ResetStep:= TRUE;
				SC_OvlStola.Step:= 23;
			ELSIF SC_OvlStola.IdleTime.Q THEN
				doStol_ODBRZDENIE:= FALSE;
				doStol_OtacajVPRED:= FALSE;
				SC_OvlStola.ResetStep:= TRUE;
				SC_OvlStola.Step:= 0;
			END_IF

            IF SC_OvlStola.AlarmTime.Q THEN
				Alarmy[31]:= TRUE;
				PoruchaOtocnyStol:= TRUE;
			END_IF

		23:
			SC_OvlStola.StepName:= '23 - Vysunutie centrovania';
			SC_OvlStola.IdleTime.PT:= T#7s;
			SC_OvlStola.AlarmTime.PT:= T#7s;
			IF Stol_Manual THEN
				SC_OvlStola.IdleTime.IN:= TRUE;
			ELSE
				SC_OvlStola.AlarmTime.IN:= TRUE;
			END_IF

			IF NOT SC_OvlStola.Switch1 THEN
				doStol_ODBRZDENIE:= FALSE;
				doStol_OtacajVPRED:= FALSE;
				Stol.OUT.CentrovanieVysunut:=1;
				Stol.OUT.CentrovanieZasunut:=0;
				SC_OvlStola.Switch1:= TRUE;
			END_IF

			IF Stol.IN.CentrovanieVysunute=1 THEN
				Stol_PrebehloOtocenie:= TRUE;
				SC_OvlStola.ResetStep:= TRUE;
				SC_OvlStola.Step:= 0;
			END_IF

	END_CASE

END_ACTION
```

### Program Logical/Program/StanicaStrihania (IEC)

#### Main.st - Init, cyclic, exit code
```iecst
PROGRAM _INIT
	T_otvorenieCentrovania.PT:=T#500ms;
END_PROGRAM

PROGRAM _CYCLIC
	T_otvorenieCentrovania();

	//Volanie podprogramov//
	OvladanieGripraNaliatku;
	OvladanieGripraStriznika;
	OvladanieOdkloneniaGriprov;
	OvladanieZdvihu;

	//Volanie funkcie SequenceControl//
	SequenceControl(SC:= SC_Strihanie);

	//Reset sekcie //
	IF Strihanie_Reset OR NOT BezpOkruhOplotenia_Aktivovany OR PoruchaStanicaStrihania THEN
		SC_Strihanie.Step:= 0;
	END_IF

	//otvaranie centrovania
	IF Vyrazanie.IN.VyrazanieJeDole=1 THEN
		T_otvorenieCentrovania.IN:=0;
	END_IF

	IF EDGEPOS (T_otvorenieCentrovania.Q=1) THEN
		T_otvorenieCentrovania.IN:=0;
		Vyrazanie.OUT.CentrovanieOtvorit:=1;
		Vyrazanie.OUT.CentrovanieZatvorit:=0;
	END_IF

	CASE SC_Strihanie.Step OF

		0:
			SC_Strihanie.StepName:='0 - Nulovanie';
			SC_OvlGripraNaliatku.Step:= 0;
			SC_OvlGripraStriznika.Step:= 0;
			SC_OvlOdklonenia.Step:= 0;
			SC_OvlZdvihu.Step:= 0;
			Strihanie_Automat:= FALSE;
			Strihanie_KoniecVyroby:= FALSE;
			Strihanie_KoniecCyklu:= FALSE;
			Strihanie_Manual:= FALSE;
			Strihanie_PoINIT:= FALSE;
			Strihanie_Reset:= FALSE;
			Strihanie_UkoncilCyklus:= FALSE;
			PocetOtvoreniGriprov:= 0;
			GriperStriznika_ZATVORENY:= FALSE;
			GriperNaliatkuZATVORENY:= FALSE;
			Strihanie_SpustiRazenie:= FALSE;
			IF BezpOkruhOplotenia_Aktivovany AND NOT PoruchaStanicaStrihania THEN
				SC_Strihanie.ResetStep:= TRUE;
				SC_Strihanie.Step:= 1;
			END_IF

		1:
			SC_Strihanie.StepName:='1 - Rozhodnutie o cinnosti';
			IF Strihanie_Automat THEN
				SC_Strihanie.Step:= 2;
			ELSIF Strihanie_Manual THEN
				SC_Strihanie.Step:= 700;
			END_IF

			//********************************************************Inicializácia****************************************************************************//
		2:
			SC_Strihanie.StepName:='2 - Inicializacia - cakanie na spustenie';
			SC_Strihanie.IdleTime.PT:= T#500ms;
			SC_Strihanie.AlarmTime.PT:= T#5s;
			SC_Strihanie.IdleTime.IN:= TRUE;

			IF SC_Strihanie.IdleTime.Q THEN
				SC_Strihanie.ResetStep:= TRUE;
				SC_Strihanie.Step:= 3;
			END_IF

		3:
			SC_Strihanie.StepName:='3 - Inicializacia - zasunutie zdvihu rotora';
			SC_Strihanie.IdleTime.PT:= T#500ms;
			SC_Strihanie.AlarmTime.PT:= T#5s;

			IF NOT SC_Strihanie.Switch1 THEN
				Rotor_POLOZ:= TRUE;
				SC_Strihanie.Switch1:= TRUE;
			END_IF

			IF Vyrazanie.IN.VyrazanieJeDole THEN
				SC_Strihanie.ResetStep:= TRUE;
				SC_Strihanie.Step:= 4;
			END_IF

		4:
			SC_Strihanie.StepName:='4 - Inicializacia -  kontrola otvorenia griprov';
			SC_Strihanie.IdleTime.PT:= T#500ms;
			SC_Strihanie.AlarmTime.PT:= T#5s;

			IF Vyrazanie.IN.UchytenieKolikaDrzimkus OR Vyrazanie.IN.UchytenieKolikaDrzimkus THEN
				SC_Strihanie.ResetStep:= TRUE;
				SC_Strihanie.Step:= 5;
			ELSIF Vyrazanie.IN.UchytenieNaliatkuOtvorene AND Vyrazanie.IN.UchytenieKolikaOtvorene THEN
				SC_Strihanie.ResetStep:= TRUE;
				SC_Strihanie.Step:= 7;
			END_IF

		5:
			SC_Strihanie.StepName:='4 - Inicializacia -  otocenie griprov do pozicie odhodenia';
			SC_Strihanie.IdleTime.PT:= T#500ms;
			SC_Strihanie.AlarmTime.PT:= T#5s;

			IF NOT SC_Strihanie.Switch1 THEN
				OdklonGriprov_ZAHODENIE:= TRUE;
				SC_Strihanie.Switch1:= TRUE;
			END_IF

			IF Vyrazanie.IN.OdhadzovanieJeVzadu THEN
				SC_Strihanie.ResetStep:= TRUE;
				SC_Strihanie.Step:= 6;
			END_IF

		6:
			SC_Strihanie.StepName:='6 - Inicializacia - otvorenie griprov';
			SC_Strihanie.IdleTime.PT:= T#500ms;
			SC_Strihanie.AlarmTime.PT:= T#5s;

			IF NOT SC_Strihanie.Switch1 THEN
				GriperNaliatku_OTVOR:= TRUE;
				GriperStriznika_OTVOR:= TRUE;
				SC_Strihanie.Switch1:= TRUE;
			END_IF

			IF Vyrazanie.IN.UchytenieKolikaOtvorene AND Vyrazanie.IN.UchytenieNaliatkuOtvorene THEN
				SC_Strihanie.ResetStep:= TRUE;
				SC_Strihanie.Step:= 7;
			END_IF

		7:
			SC_Strihanie.StepName:='7 - Inicializacia - otocenie griprov do pozicie odoberania';
			SC_Strihanie.IdleTime.PT:= T#500ms;
			SC_Strihanie.AlarmTime.PT:= T#5s;
			SC_Strihanie.IdleTime.IN:= TRUE;

			IF NOT SC_Strihanie.Switch1 AND SC_Strihanie.IdleTime.Q THEN
				OdklonGriprov_ODOBERANIE:= TRUE;
				SC_Strihanie.Switch1:= TRUE;
			END_IF

			IF Vyrazanie.IN.OdhadzovanieJeVpredu THEN
				Strihanie_PoINIT:= TRUE;
				SC_Strihanie.ResetStep:= TRUE;
				SC_Strihanie.Step:= 8;
			END_IF

		8:
			SC_Strihanie.StepName:='8 - Inicializacia - otvorenie centrovania';
			SC_Strihanie.IdleTime.PT:= T#500ms;
			SC_Strihanie.AlarmTime.PT:= T#5s;
			SC_Strihanie.IdleTime.IN:= TRUE;

			IF NOT SC_Strihanie.Switch1 AND SC_Strihanie.IdleTime.Q THEN
				Vyrazanie.OUT.CentrovanieOtvorit:= TRUE;
				Vyrazanie.OUT.CentrovanieZatvorit:= FALSE;
				SC_Strihanie.Switch1:= TRUE;
			END_IF

			IF Vyrazanie.IN.CentrovanieOtvorene THEN
				Strihanie_PoINIT:= TRUE;
				SC_Strihanie.ResetStep:= TRUE;
				SC_Strihanie.Step:= 100;
			END_IF

			//********************************************************Automatický režim****************************************************************************//
		100:
			SC_Strihanie.StepName:='100 - Automaticky rezim - cakanie na start cyklu';
			SC_Strihanie.IdleTime.PT:= T#500ms;
			SC_Strihanie.AlarmTime.PT:= T#5s;

            SC_Strihanie.IdleTime.IN:= NOT Vyrazanie.IN.KusPritomny;

			IF Strihanie_KoniecCyklu THEN
				SC_Strihanie.ResetStep:= TRUE;
				SC_Strihanie.Step:= 0;
			ELSIF Zariadenie_PrebiehaRevorkRezim THEN
				Strihanie_UkoncilCyklus:= TRUE;
                SC_Strihanie.ResetStep:= TRUE;
				SC_Strihanie.Step:= 120;
			ELSIF Stol_PoINIT AND NOT Strihanie_UkoncilCyklus AND Vyrazanie.IN.KusPritomny AND diStol_SnimacPolohyStola THEN
				SC_Strihanie.ResetStep:= TRUE;
				SC_Strihanie.Step:= 101;
			ELSIF Stol_PoINIT AND NOT Strihanie_UkoncilCyklus AND NOT Vyrazanie.IN.KusPritomny AND SC_Strihanie.IdleTime.Q AND diStol_SnimacPolohyStola THEN
				Strihanie_UkoncilCyklus:= TRUE;
                Strihanie_SpustiRazenie:= TRUE;
				SC_Strihanie.ResetStep:= TRUE;
				SC_Strihanie.Step:= 120;
			ELSIF Strihanie_KoniecVyroby AND NOT Stol_Automat THEN
				SC_Strihanie.ResetStep:= TRUE;
				SC_Strihanie.Step:= 0;
			END_IF

		101:
			SC_Strihanie.StepName:='101 - Automaticky rezim - zacentrovanie rotora';
			SC_Strihanie.IdleTime.PT:= T#500ms;
			SC_Strihanie.AlarmTime.PT:= T#5s;

			IF NOT SC_Strihanie.Switch1 THEN
				Vyrazanie.OUT.CentrovanieZatvorit:= TRUE;
				Vyrazanie.OUT.CentrovanieOtvorit:= FALSE;
				SC_Strihanie.Switch1:= TRUE;
			END_IF

			IF Vyrazanie.IN.CentrovanieZatvorene THEN
				SC_Strihanie.ResetStep:= TRUE;
				SC_Strihanie.Step:= 102; (*102*)
			END_IF

		102:
			SC_Strihanie.StepName:='102 - Automaticky rezim - zodvihnutie rotora';
			SC_Strihanie.IdleTime.PT:= T#500ms;
			SC_Strihanie.AlarmTime.PT:= T#5s;

			IF NOT SC_Strihanie.Switch1 THEN
				Rotor_ZDVIHNI:= TRUE;
				SC_Strihanie.Switch1:= TRUE;
			END_IF

			IF Vyrazanie.IN.VyrazanieJeHore AND NOT PAUZA THEN
				SC_Strihanie.ResetStep:= TRUE;
				SC_Strihanie.Step:= 103;
			END_IF

		103:
			SC_Strihanie.StepName:='103 - Automaticky rezim - zatvorenie griprov, zasunutie zdvihu rotora,otocenie griprov';
			SC_Strihanie.IdleTime.PT:= T#500ms;
			SC_Strihanie.AlarmTime.PT:= T#5s;

			IF NOT SC_Strihanie.Switch1 THEN
				GriperNaliatku_ZATVOR:= TRUE;
				GriperStriznika_ZATVOR:= TRUE;
				Strihanie_SpustiRazenie:= TRUE;
				SC_Strihanie.Switch1:= TRUE;
			END_IF

			IF Vyrazanie.IN.UchytenieKolikaDrzimkus AND Vyrazanie.IN.UchytenieNaliatkuDrzimkus THEN
				T_otvorenieCentrovania.IN:=1;
				Rotor_POLOZ:= TRUE;
				OdklonGriprov_ZAHODENIE:= TRUE;
				SC_Strihanie.ResetStep:= TRUE;
				SC_Strihanie.Step:= 104;
			END_IF

		104:
			SC_Strihanie.StepName:='104 - Automaticky rezim - vystavenie signalu ukoncenie cyklu, otvorenie griprov a zatvorenie griprov';
			SC_Strihanie.IdleTime.PT:= T#700ms;
			SC_Strihanie.AlarmTime.PT:= T#5s;

			IF EDGEPOS(Vyrazanie.IN.UchytenieKolikaOtvorene = TRUE AND Vyrazanie.IN.UchytenieNaliatkuOtvorene = TRUE) THEN
				PocetOtvoreniGriprov:= PocetOtvoreniGriprov + 1;
			END_IF

			IF EDGEPOS(Vyrazanie.IN.VyrazanieJeDole = TRUE) THEN
				IF Vyrazanie.IN.KusPritomny THEN
					Strihanie_UkoncilCyklus:= TRUE;
				ELSE
					Alarmy[48]:= TRUE;
					PoruchaStanicaStrihania:= TRUE;
				END_IF
			END_IF

			IF PocetOtvoreniGriprov <2 AND Vyrazanie.IN.OdhadzovanieJeVzadu AND Vyrazanie.IN.UchytenieKolikaZatvorene  AND SC_OvlGripraNaliatku.Step = 1 AND SC_OvlGripraStriznika.Step = 1 THEN
				GriperNaliatku_OTVOR:= TRUE;
				GriperStriznika_OTVOR:= TRUE;
				SC_Strihanie.IdleTime.IN:= TRUE;
			ELSIF PocetOtvoreniGriprov <2 AND Vyrazanie.IN.UchytenieKolikaOtvorene AND Vyrazanie.IN.UchytenieNaliatkuOtvorene AND SC_Strihanie.IdleTime.Q AND SC_OvlGripraNaliatku.Step = 1 AND SC_OvlGripraStriznika.Step = 1 THEN
				GriperNaliatku_ZATVOR:= TRUE;
				GriperStriznika_ZATVOR:= TRUE;
			ELSIF PocetOtvoreniGriprov >=2 AND Vyrazanie.IN.UchytenieKolikaOtvorene AND Vyrazanie.IN.UchytenieNaliatkuOtvorene AND Vyrazanie.IN.VyrazanieJeDole THEN
				PocetOtvoreniGriprov:= 0;
				SC_Strihanie.ResetStep:= TRUE;
				Vyrazanie.OUT.CentrovanieOtvorit:=1;
				Vyrazanie.OUT.CentrovanieZatvorit:=0;
				SC_Strihanie.Step:= 110;
			END_IF

		110:
			SC_Strihanie.StepName:='110 - Automaticky rezim - otocenie griprov do pozicie odoberania';
			SC_Strihanie.IdleTime.PT:= T#500ms;
			SC_Strihanie.AlarmTime.PT:= T#5s;
			SC_Strihanie.IdleTime.IN:= TRUE;

			IF NOT SC_Strihanie.Switch1 THEN
				OdklonGriprov_ODOBERANIE:= TRUE;
				SC_Strihanie.Switch1:= TRUE;
			END_IF

			IF Vyrazanie.IN.OdhadzovanieJeVpredu AND Vyrazanie.IN.CentrovanieOtvorene=1 AND Vyrazanie.IN.VyrazanieJeDole THEN
				SC_Strihanie.ResetStep:= TRUE;
				SC_Strihanie.Step:= 120;
			END_IF

        120:
            SC_Strihanie.StepName:='120 - Automaticky rezim - cakanie na otocenie stola';
            SC_Strihanie.IdleTime.PT:= T#500ms;
            SC_Strihanie.AlarmTime.PT:= T#5s;

            IF NOT Strihanie_UkoncilCyklus AND SC_OvlZdvihu.Step = 1  THEN
				SC_Strihanie.ResetStep:= TRUE;
				SC_Strihanie.Step:= 100;
			ELSIF Strihanie_KoniecVyroby AND NOT Stol_Automat THEN
				SC_Strihanie.ResetStep:= TRUE;
				SC_Strihanie.Step:= 0;
			ELSIF Strihanie_KoniecCyklu THEN
				SC_Strihanie.ResetStep:= TRUE;
				SC_Strihanie.Step:= 0;
			END_IF

			//********************************************************Ručný režim***********************************************************************************//
		700:
			SC_Strihanie.StepName:='700 - Rucny rezim';

        //Ovládanie otvárania centrovania rotora//
            IF Strihanie_RR_Centrovanie_OTVOR THEN
                Vyrazanie.OUT.CentrovanieZatvorit:= FALSE;
                Vyrazanie.OUT.CentrovanieOtvorit:= TRUE;
                Strihanie_RR_Centrovanie_OTVOR:= FALSE;
            ELSIF Strihanie_RR_Centrovanie_ZATVOR THEN
                Vyrazanie.OUT.CentrovanieZatvorit:= TRUE;
                Vyrazanie.OUT.CentrovanieOtvorit:= FALSE;
                Strihanie_RR_Centrovanie_ZATVOR:= FALSE;
            END_IF

	END_CASE

				END_PROGRAM

PROGRAM _EXIT
				(* Insert code here *)

				END_PROGRAM
```

#### Variables.var - Local variables
```iecst
VAR
	SC_OvlZdvihu : SequenceControlTyp;
	Rotor_ZDVIHNI : BOOL;
	Rotor_POLOZ : BOOL;
	RR_Rotor_ZDVIHNI : BOOL;
	RR_Rotor_POLOZ : BOOL;
	Rotor_POLOZ_CasOFF : BOOL;
	SC_OvlGripraNaliatku : SequenceControlTyp;
	GriperNaliatku_ZATVOR : BOOL;
	GriperNaliatku_OTVOR : BOOL;
	GriperNaliatkuZATVORENY : BOOL;
	SC_OvlGripraStriznika : SequenceControlTyp;
	GriperStriznika_ZATVOR : BOOL;
	GriperStriznika_OTVOR : BOOL;
	GriperStriznika_ZATVORENY : BOOL;
	SC_OvlOdklonenia : SequenceControlTyp;
	OdklonGriprov_ODOBERANIE : BOOL;
	OdklonGriprov_ZAHODENIE : BOOL;
	PrazdnaPozicia : BOOL;
	ChybaVystrihnutia : BOOL;
	PocetOtvoreniGriprov : USINT;
	T_otvorenieCentrovania : TON;
	PAUZA : BOOL;
END_VAR
```

#### OvladanieZdvihu.st
```iecst
ACTION OvladanieZdvihu:

	//Volanie funkcie SequenceControl//
	SequenceControl(SC:= SC_OvlZdvihu);

	CASE SC_OvlZdvihu.Step OF

		0:
			SC_OvlZdvihu.StepName:= '0 - Nulovanie';
			Rotor_ZDVIHNI:= FALSE;
			Rotor_POLOZ:= FALSE;
			RR_Rotor_ZDVIHNI:= FALSE;
			RR_Rotor_POLOZ:= FALSE;
			Vyrazanie.OUT.VyrazanieVysunut:= FALSE;
			Vyrazanie.OUT.VyrazanieZasunut:= FALSE;
			ChybaVystrihnutia:= FALSE;
			IF SC_Strihanie.Step <> 0 THEN
				SC_OvlZdvihu.ResetStep:= TRUE;
				SC_OvlZdvihu.Step:= 1;
			END_IF

		1:
			SC_OvlZdvihu.StepName:= '1 - Rozhodnutie o cinnosti';
			IF Rotor_ZDVIHNI THEN
				SC_OvlZdvihu.Step:= 10;
			ELSIF Rotor_POLOZ THEN
				SC_OvlZdvihu.Step:= 20;
			ELSIF RR_Rotor_ZDVIHNI THEN
				SC_OvlZdvihu.Step:= 30;
			ELSIF RR_Rotor_POLOZ THEN
				SC_OvlZdvihu.Step:= 40;
			END_IF

		10:
			SC_OvlZdvihu.StepName:= '10 - Zodvihnutie rotora';
			SC_OvlZdvihu.IdleTime.PT:= T#8s;
			SC_OvlZdvihu.AlarmTime.PT:= T#6s;

			IF Strihanie_Manual THEN
				SC_OvlZdvihu.IdleTime.IN:= TRUE;
			ELSE
				SC_OvlZdvihu.AlarmTime.IN:= TRUE;
			END_IF

			IF NOT SC_OvlZdvihu.Switch1 THEN
				Vyrazanie.OUT.VyrazanieZasunut:= FALSE;
				Vyrazanie.OUT.VyrazanieVysunut:= TRUE;
				SC_OvlZdvihu.Switch1:= TRUE;
			END_IF

			IF SC_OvlZdvihu.AlarmTime.Q THEN
				ChybaVystrihnutia:= TRUE;
			END_IF

			IF ChybaVystrihnutia THEN
				SC_OvlZdvihu.ResetStep:= TRUE;
				SC_OvlZdvihu.Step:= 20;
			ELSIF Vyrazanie.IN.VyrazanieJeHore OR SC_OvlZdvihu.IdleTime.Q THEN
				SC_OvlZdvihu.ResetStep:= TRUE;
				SC_OvlZdvihu.Step:= 0;
			END_IF

		20:
			SC_OvlZdvihu.StepName:= '20 - Polozenie rotora';
			SC_OvlZdvihu.IdleTime.PT:= T#6s;
			SC_OvlZdvihu.AlarmTime.PT:= T#5s;

			IF Strihanie_Manual THEN
				SC_OvlZdvihu.IdleTime.IN:= TRUE;
			ELSE
				SC_OvlZdvihu.AlarmTime.IN:= TRUE;
			END_IF

			IF NOT SC_OvlZdvihu.Switch1 THEN
				Vyrazanie.OUT.VyrazanieVysunut:= FALSE;
				Vyrazanie.OUT.VyrazanieZasunut:= TRUE;
				SC_OvlZdvihu.Switch1:= TRUE;
			END_IF

			IF SC_OvlZdvihu.AlarmTime.Q THEN
				Alarmy[41]:= TRUE;
				PoruchaStanicaStrihania:= TRUE;
			END_IF

			IF ChybaVystrihnutia AND Vyrazanie.IN.VyrazanieJeDole THEN
				Alarmy[40]:= TRUE;
				PoruchaStanicaStrihania:= TRUE;
			ELSIF Vyrazanie.IN.VyrazanieJeDole OR SC_OvlZdvihu.IdleTime.Q THEN
				SC_OvlZdvihu.ResetStep:= TRUE;
				SC_OvlZdvihu.Step:= 0;
			END_IF

		30:
			SC_OvlZdvihu.StepName:= '30 - Zodvihnutie rotora v rucnom rezime';
			SC_OvlZdvihu.IdleTime.PT:= T#6s;
			SC_OvlZdvihu.AlarmTime.PT:= T#6s;

			IF NOT SC_OvlZdvihu.Switch1 THEN
				Vyrazanie.OUT.VyrazanieZasunut:= FALSE;
				Vyrazanie.OUT.VyrazanieVysunut:= TRUE;
				SC_OvlZdvihu.Switch1:= TRUE;
			END_IF

			IF Vyrazanie.IN.VyrazanieJeHore OR NOT RR_Rotor_ZDVIHNI THEN
				SC_OvlZdvihu.ResetStep:= TRUE;
				SC_OvlZdvihu.Step:= 0;
			END_IF

		40:
			SC_OvlZdvihu.StepName:= '40 - Polozenie rotora v rucnom rezime';
			SC_OvlZdvihu.IdleTime.PT:= T#6s;
			SC_OvlZdvihu.AlarmTime.PT:= T#5s;
			SC_OvlZdvihu.IdleTime.IN:= TRUE;

			IF NOT SC_OvlZdvihu.Switch1 THEN
				Vyrazanie.OUT.VyrazanieVysunut:= FALSE;
				Vyrazanie.OUT.VyrazanieZasunut:= TRUE;
				SC_OvlZdvihu.Switch1:= TRUE;
			END_IF

			IF SC_OvlZdvihu.IdleTime.Q OR Vyrazanie.IN.VyrazanieJeDole THEN
				SC_OvlZdvihu.ResetStep:= TRUE;
				SC_OvlZdvihu.Step:= 0;
			END_IF

	END_CASE

END_ACTION
```

#### OvladanieGripraNaliatku.st
```iecst
ACTION OvladanieGripraNaliatku:

	//Volanie funkcie SequenceControl//
	SequenceControl(SC:= SC_OvlGripraNaliatku);

	CASE SC_OvlGripraNaliatku.Step OF
		0:
			SC_OvlGripraNaliatku.StepName:= '0 - Nulovanie';
			GriperNaliatku_OTVOR:= FALSE;
			GriperNaliatku_ZATVOR:= FALSE;
			Vyrazanie.OUT.UchytenieNaliatkuOtvorit:= FALSE;
			Vyrazanie.OUT.UchytenieNaliatkuZatvorit:= FALSE;
			IF SC_Strihanie.Step <> 0 THEN
				SC_OvlGripraNaliatku.ResetStep:= TRUE;
				SC_OvlGripraNaliatku.Step:= 1;
			END_IF

		1:
			SC_OvlGripraNaliatku.StepName:= '1 - Rozhodnutie o cinnosti';
			IF GriperNaliatku_OTVOR THEN
				SC_OvlGripraNaliatku.Step:= 10;
			ELSIF GriperNaliatku_ZATVOR THEN
				SC_OvlGripraNaliatku.Step:= 20;
			END_IF

		10:
			SC_OvlGripraNaliatku.StepName:= '10 - Otvorenie gripra';
			SC_OvlGripraNaliatku.IdleTime.PT:= T#3s;
			SC_OvlGripraNaliatku.AlarmTime.PT:= T#3s;

			IF Strihanie_Manual THEN
				SC_OvlGripraNaliatku.IdleTime.IN:= TRUE;
			ELSE
				SC_OvlGripraNaliatku.AlarmTime.IN:= TRUE;
			END_IF

			IF NOT SC_OvlGripraNaliatku.Switch1 THEN
				Vyrazanie.OUT.UchytenieNaliatkuOtvorit:= TRUE;
				SC_OvlGripraNaliatku.Switch1:= TRUE;
			END_IF

			IF SC_OvlGripraNaliatku.AlarmTime.Q THEN
				Alarmy[42]:= TRUE;
				PoruchaStanicaStrihania:= TRUE;
			END_IF

			IF Vyrazanie.IN.UchytenieNaliatkuOtvorene OR SC_OvlGripraNaliatku.IdleTime.Q THEN
				SC_OvlGripraNaliatku.ResetStep:= TRUE;
				SC_OvlGripraNaliatku.Step:= 0;
			END_IF

		20:
			SC_OvlGripraNaliatku.StepName:= '20 - Zatvorenie gripra';
			SC_OvlGripraNaliatku.IdleTime.PT:= T#3s;
			SC_OvlGripraNaliatku.AlarmTime.PT:= T#3s;

			IF Strihanie_Manual THEN
				SC_OvlGripraNaliatku.IdleTime.IN:= TRUE;
			ELSE
				SC_OvlGripraNaliatku.AlarmTime.IN:= TRUE;
			END_IF

			IF NOT SC_OvlGripraNaliatku.Switch1 THEN
				Vyrazanie.OUT.UchytenieNaliatkuZatvorit:= TRUE;
				SC_OvlGripraNaliatku.Switch1:= TRUE;
			END_IF

			IF SC_OvlGripraNaliatku.AlarmTime.Q THEN
				Alarmy[43]:= TRUE;
				PoruchaStanicaStrihania:= TRUE;
			END_IF

			IF (Vyrazanie.IN.UchytenieNaliatkuDrzimkus OR Vyrazanie.IN.UchytenieKolikaDrzimkus) OR SC_OvlGripraNaliatku.IdleTime.Q THEN
				SC_OvlGripraNaliatku.ResetStep:= TRUE;
				SC_OvlGripraNaliatku.Step:= 0;
			END_IF

	END_CASE

			END_ACTION
```

#### OvladanieGripraStriznika.st
```iecst
ACTION OvladanieGripraStriznika:

	//Volanie funkcie SequenceControl//
	SequenceControl(SC:= SC_OvlGripraStriznika);

	CASE SC_OvlGripraStriznika.Step OF
		0:
			SC_OvlGripraStriznika.StepName:= '0 - Nulovanie';
			GriperStriznika_OTVOR:= FALSE;
			GriperStriznika_ZATVOR:= FALSE;
			Vyrazanie.OUT.UchytenieKolikaOtvorit:= FALSE;
			Vyrazanie.OUT.UchytenieKolikaZatvorit:= FALSE;
			IF SC_Strihanie.Step <> 0 THEN
				SC_OvlGripraStriznika.ResetStep:= TRUE;
				SC_OvlGripraStriznika.Step:= 1;
			END_IF

		1:
			SC_OvlGripraStriznika.StepName:= '1 - Rozhodnutie o cinnosti';
			IF GriperStriznika_OTVOR THEN
				SC_OvlGripraStriznika.Step:= 10;
			ELSIF GriperStriznika_ZATVOR THEN
				SC_OvlGripraStriznika.Step:= 20;
			END_IF

		10:
			SC_OvlGripraStriznika.StepName:= '10 - Otvorenie gripra';
			SC_OvlGripraStriznika.IdleTime.PT:= T#3s;
			SC_OvlGripraStriznika.AlarmTime.PT:= T#3s;

			IF Strihanie_Manual THEN
				SC_OvlGripraStriznika.IdleTime.IN:= TRUE;
			ELSE
				SC_OvlGripraStriznika.AlarmTime.IN:= TRUE;
			END_IF

			IF NOT SC_OvlGripraStriznika.Switch1 THEN
				Vyrazanie.OUT.UchytenieKolikaOtvorit:= TRUE;
				SC_OvlGripraStriznika.Switch1:= TRUE;
			END_IF

			IF SC_OvlGripraStriznika.AlarmTime.Q THEN
				Alarmy[44]:= TRUE;
				PoruchaStanicaStrihania:= TRUE;
			END_IF

			IF Vyrazanie.IN.UchytenieKolikaOtvorene OR SC_OvlGripraStriznika.IdleTime.Q THEN
				SC_OvlGripraStriznika.ResetStep:= TRUE;
				SC_OvlGripraStriznika.Step:= 0;
			END_IF

		20:
			SC_OvlGripraStriznika.StepName:= '20 - Zatvorenie gripra';
			SC_OvlGripraStriznika.IdleTime.PT:= T#3s;
			SC_OvlGripraStriznika.AlarmTime.PT:= T#3s;

			IF Strihanie_Manual THEN
				SC_OvlGripraStriznika.IdleTime.IN:= TRUE;
			ELSE
				SC_OvlGripraStriznika.AlarmTime.IN:= TRUE;
			END_IF

			IF NOT SC_OvlGripraStriznika.Switch1 THEN
				Vyrazanie.OUT.UchytenieKolikaZatvorit:= TRUE;
				SC_OvlGripraStriznika.Switch1:= TRUE;
			END_IF

			IF SC_OvlGripraStriznika.AlarmTime.Q THEN
				Alarmy[45]:= TRUE;
				PoruchaStanicaStrihania:= TRUE;
			END_IF

			IF Vyrazanie.IN.UchytenieKolikaDrzimkus OR SC_OvlGripraStriznika.IdleTime.Q THEN
				SC_OvlGripraStriznika.ResetStep:= TRUE;
				SC_OvlGripraStriznika.Step:= 0;
			END_IF

	END_CASE

END_ACTION
```

#### OvladanieOdkloneniaGriprov.st
```iecst
ACTION OvladanieOdkloneniaGriprov:

	//Volanie funkcie SequenceControl//
	SequenceControl(SC:= SC_OvlOdklonenia);

	CASE SC_OvlOdklonenia.Step OF

		0:
			SC_OvlOdklonenia.StepName:= '0 - Nulovanie';
			OdklonGriprov_ODOBERANIE:= FALSE;
			OdklonGriprov_ZAHODENIE:= FALSE;
			Vyrazanie.OUT.OdhadzovanieVysunut:= FALSE;
			Vyrazanie.OUT.OdhadzovanieZasunut:= FALSE;
			IF SC_Strihanie.Step <> 0 THEN
				SC_OvlOdklonenia.ResetStep:= TRUE;
				SC_OvlOdklonenia.Step:= 1;
			END_IF

		1:
			SC_OvlOdklonenia.StepName:= '1 - Rozhodnutie o cinnosti';
			IF OdklonGriprov_ODOBERANIE THEN
				SC_OvlOdklonenia.Step:= 10;
			ELSIF OdklonGriprov_ZAHODENIE THEN
				SC_OvlOdklonenia.Step:= 20;
			END_IF

		10:
			SC_OvlOdklonenia.StepName:= '10 - Odklopenie griprov do pozicie odoberania';
			SC_OvlOdklonenia.IdleTime.PT:= T#3s;
			SC_OvlOdklonenia.AlarmTime.PT:= T#7s;

			IF Strihanie_Manual THEN
				SC_OvlOdklonenia.IdleTime.IN:= TRUE;
			ELSE
				SC_OvlOdklonenia.AlarmTime.IN:= TRUE;
			END_IF

			IF NOT SC_OvlOdklonenia.Switch1 THEN
				Vyrazanie.OUT.OdhadzovanieVysunut:= TRUE;
				SC_OvlOdklonenia.Switch1:= TRUE;
			END_IF

			IF SC_OvlOdklonenia.AlarmTime.Q THEN
				Alarmy[46]:= TRUE;
				PoruchaStanicaStrihania:= TRUE;
			END_IF

			IF (Vyrazanie.IN.OdhadzovanieJeVpredu AND Vyrazanie.IN.OdhadzovanieJeVpredu2) OR SC_OvlOdklonenia.IdleTime.Q THEN
				SC_OvlOdklonenia.ResetStep:= TRUE;
				SC_OvlOdklonenia.Step:= 0;
			END_IF

		20:
			SC_OvlOdklonenia.StepName:= '20 - Odklopenie griprov do pozicie zahodenia';
			SC_OvlOdklonenia.IdleTime.PT:= T#3s;
			SC_OvlOdklonenia.AlarmTime.PT:= T#7s;

			IF Strihanie_Manual THEN
				SC_OvlOdklonenia.IdleTime.IN:= TRUE;
			ELSE
				SC_OvlOdklonenia.AlarmTime.IN:= TRUE;
			END_IF

			IF NOT SC_OvlOdklonenia.Switch1 THEN
				Vyrazanie.OUT.OdhadzovanieZasunut:= TRUE;
				SC_OvlOdklonenia.Switch1:= TRUE;
			END_IF

			IF SC_OvlOdklonenia.AlarmTime.Q THEN
				Alarmy[47]:= TRUE;
				PoruchaStanicaStrihania:= TRUE;
			END_IF

			IF Vyrazanie.IN.OdhadzovanieJeVzadu OR SC_OvlOdklonenia.IdleTime.Q THEN
				SC_OvlOdklonenia.ResetStep:= TRUE;
				SC_OvlOdklonenia.Step:= 0;
			END_IF

	END_CASE

END_ACTION
```

### Program Logical/Program/StanicaRazenia (IEC)

#### Main.st - Init, cyclic, exit code
```iecst
PROGRAM _INIT
	(* Insert code here *)

END_PROGRAM

PROGRAM _CYCLIC

	//Volanie podprogramov//
	OvladanieZdvihu;

	//Volanie funkcie SequenceControl//
	SequenceControl(SC:= SC_Razenie);

	//Prepočet času razenia//
	CasRazenia:= REAL_TO_TIME(TP_Razenie_CasRazenia * 1000);

	//Reset sekcie //
	IF Razenie_Reset OR NOT BezpOkruhOplotenia_Aktivovany OR PoruchaStanicaRazenia THEN
		SC_Razenie.Step:= 0;
	END_IF

	CASE SC_Razenie.Step OF

		0:
			SC_Razenie.StepName:='0 - Nulovanie';
			SC_OvlZdvihu.Step:= 0;
			Razenie_Automat:= FALSE;
			Razenie_KoniecVyroby:= FALSE;
			Razenie_KoniecCyklu:= FALSE;
			Razenie_Manual:= FALSE;
			Razenie_PoINIT:= FALSE;
			Razenie_Reset:= FALSE;
			Razenie_UkoncilCyklus:= FALSE;
			Strihanie_StavBUSY:= FALSE;
			Zdvih_Napolohovany:= FALSE;
			IF BezpOkruhOplotenia_Aktivovany AND NOT PoruchaStanicaRazenia THEN
				SC_Razenie.ResetStep:= TRUE;
				SC_Razenie.Step:= 1;
			END_IF

		1:
			SC_Razenie.StepName:='1 - Rozhodnutie o cinnosti';
			IF Razenie_Automat THEN
				SC_Razenie.Step:= 2;
			ELSIF Razenie_Manual THEN
				SC_Razenie.Step:= 700;
			END_IF

			//********************************************************Inicializácia****************************************************************************//

		2:
			SC_Razenie.StepName:='2 - Inicializacia - cakanie na spustenie';
			SC_Razenie.IdleTime.PT:= T#500ms;
			SC_Razenie.AlarmTime.PT:= T#5s;
			SC_Razenie.IdleTime.IN:= TRUE;

			IF SC_Razenie.IdleTime.Q THEN
				SC_Razenie.ResetStep:= TRUE;
				SC_Razenie.Step:= 3;
			END_IF

		3:
			SC_Razenie.StepName:='3 - Inicializacia - zasunutie zdvihu';
			SC_Razenie.IdleTime.PT:= T#500ms;
			SC_Razenie.AlarmTime.PT:= T#5s;

			IF NOT SC_Razenie.Switch1 THEN
				Rotor_POLOZ:= TRUE;
				SC_Razenie.Switch1:= TRUE;
			END_IF

			IF diRazenie_ZdvihSpodnaPoloha THEN
				Razenie_PoINIT:= TRUE;
				SC_Razenie.ResetStep:= TRUE;
				SC_Razenie.Step:= 100;
			END_IF

			//********************************************************Automatický režim****************************************************************************//
		100:
			SC_Razenie.StepName:='100 - Automaticky rezim - cakanie na start cyklu';
			SC_Razenie.IdleTime.PT:= T#500ms;
			SC_Razenie.AlarmTime.PT:= T#5s;

			SC_Razenie.IdleTime.IN:= NOT diRazenie_PritomnostRotora;

			IF Razenie_KoniecCyklu THEN
				SC_Razenie.ResetStep:= TRUE;
				SC_Razenie.Step:= 0;
			ELSIF Zariadenie_PrebiehaRevorkRezim THEN
				SC_Razenie.ResetStep:= TRUE;
				SC_Razenie.Step:= 120;
			ELSIF Stol_PoINIT AND NOT Razenie_UkoncilCyklus AND diRazenie_PritomnostRotora AND diStol_SnimacPolohyStola (*AND Strihanie_SpustiRazenie*) THEN
				Strihanie_StavBUSY:= FALSE;
				Strihanie_SpustiRazenie:= FALSE;
				SC_Razenie.ResetStep:= TRUE;
				SC_Razenie.Step:= 101;//101
			ELSIF Stol_PoINIT AND NOT Razenie_UkoncilCyklus AND NOT diRazenie_PritomnostRotora AND SC_Razenie.IdleTime.Q AND diStol_SnimacPolohyStola THEN
				Strihanie_StavBUSY:= FALSE;
				SC_Razenie.ResetStep:= TRUE;
				SC_Razenie.Step:= 120;
			ELSIF Razenie_KoniecVyroby AND NOT Stol_Automat THEN
				SC_Razenie.ResetStep:= TRUE;
				SC_Razenie.Step:= 0;
			END_IF

		101:
			SC_Razenie.StepName:='101 - Automaticky rezim - zodvihnutie rotora';
			SC_Razenie.IdleTime.PT:= T#500ms;
			SC_Razenie.AlarmTime.PT:= T#5s;

			IF NOT SC_Razenie.Switch1 AND SC_OvlZdvihu.Step = 1 THEN
				Rotor_ZDVIHNI:= TRUE;
				SC_Razenie.Switch1:= TRUE;
			END_IF

			IF Zdvih_Napolohovany THEN
				Zdvih_Napolohovany:= FALSE;
				SC_Razenie.ResetStep:= TRUE;
				SC_Razenie.Step:= 103;
			END_IF

		103:
			SC_Razenie.StepName:='103 - Automaticky rezim - zasunutie zdvihu';
			SC_Razenie.IdleTime.PT:= T#500ms;
			SC_Razenie.AlarmTime.PT:= T#5s;

			IF NOT SC_Razenie.Switch1 AND SC_OvlZdvihu.Step = 1 THEN
				Rotor_POLOZ:= TRUE;
				SC_Razenie.Switch1:= TRUE;
			END_IF

			IF diRazenie_ZdvihSpodnaPoloha AND diRazenie_PritomnostRotora THEN
				SC_Razenie.ResetStep:= TRUE;
				SC_Razenie.Step:= 120;
			ELSIF diRazenie_ZdvihSpodnaPoloha AND NOT diRazenie_PritomnostRotora THEN
				Alarmy[52]:= TRUE;
				PoruchaStanicaRazenia:= TRUE;
			END_IF

		120:
			SC_Razenie.StepName:='120 - Automaticky rezim - vystavenie signalu ukoncenie pracovneho cyklu';
			SC_Razenie.IdleTime.PT:= T#500ms;
			SC_Razenie.AlarmTime.PT:= T#5s;

			IF diRazenie_ZdvihSpodnaPoloha THEN
				Razenie_UkoncilCyklus:= TRUE;
				SC_Razenie.ResetStep:= TRUE;
				SC_Razenie.Step:= 121;
			END_IF

		121:
			SC_Razenie.StepName:='121 - Automaticky rezim - cakanie na otocenie stola';
			SC_Razenie.IdleTime.PT:= T#500ms;
			SC_Razenie.AlarmTime.PT:= T#5s;

			IF NOT Razenie_UkoncilCyklus AND SC_OvlZdvihu.Step = 1 THEN
				SC_Razenie.ResetStep:= TRUE;
				SC_Razenie.Step:= 100;
			ELSIF Razenie_KoniecVyroby AND NOT Stol_Automat THEN
				SC_Razenie.ResetStep:= TRUE;
				SC_Razenie.Step:= 0;
			ELSIF Razenie_KoniecCyklu THEN
				SC_Razenie.ResetStep:= TRUE;
				SC_Razenie.Step:= 0;
			END_IF

			//********************************************************Ručný režim***********************************************************************************//
		700:
			SC_Razenie.StepName:='700 - Rucny rezim';

	END_CASE
END_PROGRAM

PROGRAM _EXIT
END_PROGRAM
```

#### Variables.var - Local variables
```iecst
VAR
	SC_OvlZdvihu : SequenceControlTyp;
	Rotor_ZDVIHNI : BOOL;
	Rotor_POLOZ : BOOL;
	Rotor_POLOZ_CasOFF : BOOL;
	RR_Rotor_ZDVIHNI : BOOL;
	CasRazenia : TIME;
	Strihanie_StavBUSY : BOOL;
	PrazdnaPozicia : BOOL;
	Zdvih_Napolohovany : BOOL;
END_VAR
```

#### OvladanieZdvihu.st
```iecst
ACTION OvladanieZdvihu:

	//Volanie funkcie SequenceControl//
	SequenceControl(SC:= SC_OvlZdvihu);

	CASE SC_OvlZdvihu.Step OF

		0:
			SC_OvlZdvihu.StepName:= '0 - Nulovanie';
			Rotor_ZDVIHNI:= FALSE;
			Rotor_POLOZ:= FALSE;
			Rotor_POLOZ_CasOFF:= FALSE;
			RR_Rotor_ZDVIHNI:= FALSE;
			doRazenie_ZdvihRotora:= FALSE;
			doRazenie_ZostupRotora:= FALSE;
			IF SC_Razenie.Step <> 0 THEN
				SC_OvlZdvihu.ResetStep:= TRUE;
				SC_OvlZdvihu.Step:= 1;
			END_IF

		1:
			SC_OvlZdvihu.StepName:= '1 - Rozhodnutie o cinnosti';
			IF Rotor_ZDVIHNI THEN
				SC_OvlZdvihu.Step:= 10;
			ELSIF Rotor_POLOZ THEN
				SC_OvlZdvihu.Step:= 20;
			ELSIF RR_Rotor_ZDVIHNI THEN
				SC_OvlZdvihu.Step:= 30;
			ELSIF Rotor_POLOZ_CasOFF THEN
				SC_OvlZdvihu.Step:= 40;
			END_IF

		10:
			SC_OvlZdvihu.StepName:= '10 - Zodvihnutie rotora';
			IF Razenie_Automat THEN
				SC_OvlZdvihu.IdleTime.PT:= T#500ms;
			ELSIF Razenie_Manual THEN
				SC_OvlZdvihu.IdleTime.PT:= T#6s;
			END_IF
			SC_OvlZdvihu.AlarmTime.PT:= T#6s;

			IF Razenie_Automat THEN
				SC_OvlZdvihu.AlarmTime.IN:= TRUE;
				IF diRazenie_ZdvihHornaPoloha THEN
					SC_OvlZdvihu.IdleTime.IN:= TRUE;
				END_IF
			ELSIF Razenie_Manual THEN
				SC_OvlZdvihu.IdleTime.IN:= TRUE;
			END_IF

			IF NOT SC_OvlZdvihu.Switch1 THEN
				doRazenie_ZostupRotora:= FALSE;
				doRazenie_ZdvihRotora:= TRUE;
				SC_OvlZdvihu.Switch1:= TRUE;
			END_IF

			IF SC_OvlZdvihu.AlarmTime.Q THEN
				Alarmy[50]:= TRUE;
				PoruchaStanicaRazenia:= TRUE;
			END_IF

			IF SC_OvlZdvihu.IdleTime.Q THEN
				Zdvih_Napolohovany:= TRUE;
				SC_OvlZdvihu.ResetStep:= TRUE;
				SC_OvlZdvihu.Step:= 0;
			END_IF

		20:
			SC_OvlZdvihu.StepName:= '20 - Polozenie rotora';
			SC_OvlZdvihu.IdleTime.PT:= T#6s;
			SC_OvlZdvihu.AlarmTime.PT:= T#6s;

			IF Razenie_Manual THEN
				SC_OvlZdvihu.IdleTime.IN:= TRUE;
			ELSE
				SC_OvlZdvihu.AlarmTime.IN:= TRUE;
			END_IF

			IF NOT SC_OvlZdvihu.Switch1 THEN
				doRazenie_ZdvihRotora:= FALSE;
				doRazenie_ZostupRotora:= TRUE;
				SC_OvlZdvihu.Switch1:= TRUE;
			END_IF

			IF SC_OvlZdvihu.AlarmTime.Q THEN
				Alarmy[51]:= TRUE;
				PoruchaStanicaRazenia:= TRUE;
			END_IF

			IF diRazenie_ZdvihSpodnaPoloha OR SC_OvlZdvihu.IdleTime.Q THEN
				SC_OvlZdvihu.ResetStep:= TRUE;
				SC_OvlZdvihu.Step:= 0;
			END_IF

		30:
			SC_OvlZdvihu.StepName:= '30 - Zodvihnutie rotora v rucnom rezime';
			SC_OvlZdvihu.IdleTime.PT:= T#6s;
			SC_OvlZdvihu.AlarmTime.PT:= T#6s;

			IF NOT SC_OvlZdvihu.Switch1 THEN
				doRazenie_ZostupRotora:= FALSE;
				doRazenie_ZdvihRotora:= TRUE;
				SC_OvlZdvihu.Switch1:= TRUE;
			END_IF

			IF diRazenie_ZdvihHornaPoloha OR NOT RR_Rotor_ZDVIHNI THEN
				doRazenie_ZostupRotora:= FALSE;
				doRazenie_ZdvihRotora:= FALSE;
				SC_OvlZdvihu.ResetStep:= TRUE;
				SC_OvlZdvihu.Step:= 0;
			END_IF

		40:
			SC_OvlZdvihu.StepName:= '40 - Polozenie rotora';
			SC_OvlZdvihu.IdleTime.PT:= T#3s;
			SC_OvlZdvihu.AlarmTime.PT:= T#6s;
			SC_OvlZdvihu.IdleTime.IN:= TRUE;

			IF NOT SC_OvlZdvihu.Switch1 THEN
				doRazenie_ZdvihRotora:= FALSE;
				doRazenie_ZostupRotora:= TRUE;
				SC_OvlZdvihu.Switch1:= TRUE;
			END_IF

			IF SC_OvlZdvihu.IdleTime.Q THEN
				SC_OvlZdvihu.ResetStep:= TRUE;
				SC_OvlZdvihu.Step:= 0;
			END_IF

	END_CASE

END_ACTION
```

### Program Logical/Program/StanicaVnutornehoValcovania (IEC)

#### Main.st - Init, cyclic, exit code
```iecst
PROGRAM _INIT
	(* Insert code here *)

END_PROGRAM

PROGRAM _CYCLIC

	//Volanie podprogramov//
	OvladanieGripra;
	OvladanieOtacaniaRotora;
	OvladanieZdvihuRotora;
	OvladanieZdvihuServa;

	//Volanie funkcie SequenceControl//
	SequenceControl(SC:= SC_Valcovanie);

	//Prepočet času streku oleja//
	CasStrekuOleja:= REAL_TO_TIME(TP_Valcovanie_CasStrekuOleja * 1000);

	//Prepočet času valcovania//
	CasValcovania_ms:= REAL_TO_TIME(TP_CasValcovania_s * 1000);

	//Striekanie oleja//
	IF doValcovanie_DavkaOleja THEN
		CasStrikaniaOleja.IN:= TRUE;
	END_IF

	IF CasStrikaniaOleja.Q THEN
		CasStrikaniaOleja.IN:= FALSE;
		doValcovanie_DavkaOleja:= FALSE;
	END_IF

	CasStrikaniaOleja.PT:= CasStrekuOleja;
	CasStrikaniaOleja();

	//Reset sekcie //
	IF Valcovanie_Reset OR NOT BezpOkruhOplotenia_Aktivovany OR PoruchaStanicaValcovania THEN
		SC_Valcovanie.Step:= 0;
	END_IF

	CASE SC_Valcovanie.Step OF

		0:
			SC_Valcovanie.StepName:='0 - Nulovanie';
			SC_OvlGripra.Step:= 0;
			SC_OvlOtacania.Step:= 0;
			SC_OvlServoZdvihu.Step:= 0;
			SC_OvlZdvihu.Step:= 0;
			Valcovanie_Automat:= FALSE;
			Valcovanie_KoniecVyroby:= FALSE;
			Valcovanie_KoniecCyklu:= FALSE;
			Valcovanie_Manual:= FALSE;
			Valcovanie_PoINIT:= FALSE;
			Valcovanie_Reset:= FALSE;
			Valcovanie_ZdvihVPOZICI:= FALSE;
			Valcovanie_UkoncilCyklus:= FALSE;
			doValcovanie_DavkaOleja:= FALSE;
			PocetCyklovValcovania:= 0;
			RR_StartOlejovania:= FALSE;
			RR_PoziciaValcovania:= FALSE;
			RR_PoziciaVychodzia:= FALSE;
			Priznak_ValcovanieNG:= FALSE;
			Priznak_ValcovanieOK:= FALSE;
			IF BezpOkruhOplotenia_Aktivovany AND NOT PoruchaStanicaValcovania THEN
				SC_Valcovanie.ResetStep:= TRUE;
				SC_Valcovanie.Step:= 1;
			END_IF

		1:
			SC_Valcovanie.StepName:='1 - Rozhodnutie o cinnosti';
			IF Valcovanie_Automat THEN
				SC_Valcovanie.Step:= 2;
			ELSIF Valcovanie_Manual THEN
				SC_Valcovanie.Step:= 700;
			END_IF

			//********************************************************Inicializácia****************************************************************************//

		2:
			SC_Valcovanie.StepName:='2 - Inicializacia - cakanie na spustenie';
			SC_Valcovanie.IdleTime.PT:= T#500ms;
			SC_Valcovanie.AlarmTime.PT:= T#5s;
			SC_Valcovanie.IdleTime.IN:= TRUE;

			IF SC_Valcovanie.IdleTime.Q THEN
				SC_Valcovanie.ResetStep:= TRUE;
				SC_Valcovanie.Step:= 3;
			END_IF

		3:
			SC_Valcovanie.StepName:='3 - Inicializacia - kontrola home serva zdvihu';
			SC_Valcovanie.IdleTime.PT:= T#500ms;
			SC_Valcovanie.AlarmTime.PT:= T#5s;

			IF Motion[3].status.DriveStatus.HomingOk THEN
				SC_Valcovanie.ResetStep:= TRUE;
				SC_Valcovanie.Step:= 5;
			ELSE
				SC_Valcovanie.ResetStep:= TRUE;
				SC_Valcovanie.Step:= 4;
			END_IF

		4:
			SC_Valcovanie.StepName:='4 - Inicializacia - homing serva zdvihu';
			SC_Valcovanie.IdleTime.PT:= T#500ms;
			SC_Valcovanie.AlarmTime.PT:= T#5s;

			IF NOT SC_Valcovanie.Switch1 THEN
				Valcovanie_ZdvihHOME:= TRUE;
				SC_Valcovanie.Switch1:= TRUE;
			END_IF

			IF Motion[3].status.DriveStatus.HomingOk THEN
				SC_Valcovanie.IdleTime.IN:= TRUE;
			END_IF

			IF Motion[3].status.DriveStatus.HomingOk AND SC_Valcovanie.IdleTime.Q AND Motion[3].state.StandStill THEN
				SC_Valcovanie.ResetStep:= TRUE;
				SC_Valcovanie.Step:= 5;
			END_IF

		5:
			SC_Valcovanie.StepName:='5 - Inicializacia - otvorenie gripra';
			SC_Valcovanie.IdleTime.PT:= T#500ms;
			SC_Valcovanie.AlarmTime.PT:= T#5s;

			IF NOT SC_Valcovanie.Switch1 THEN
				Otvor_Griper:= TRUE;
				SC_Valcovanie.Switch1:= TRUE;
			END_IF

			IF diValcovanie_GriperOtvoreny THEN
				SC_Valcovanie.ResetStep:= TRUE;
				SC_Valcovanie.Step:= 6;
			END_IF

		6:
			SC_Valcovanie.StepName:='6 - Inicializacia - zdvih motora do vychodiskovej pozicie, zasunutie zdvihu rotora';
			SC_Valcovanie.IdleTime.PT:= T#500ms;
			SC_Valcovanie.AlarmTime.PT:= T#5s;

			Valcovanie_ZadanaPozMM:= 15;

			IF NOT SC_Valcovanie.Switch1 THEN
				ServoZdvih_Polohuj:= TRUE;
				Rotor_POLOZ:= TRUE;
				SC_Valcovanie.Switch1:= TRUE;
			END_IF

			IF diValcovanie_ZdvihSpodnaPoloha AND Valcovanie_ZdvihVPOZICI THEN
				Valcovanie_ZdvihVPOZICI:= FALSE;
				Valcovanie_PoINIT:= TRUE;
				SC_Valcovanie.ResetStep:= TRUE;
				SC_Valcovanie.Step:= 100;
			END_IF

			//********************************************************Automatický režim****************************************************************************//
		100:
			SC_Valcovanie.StepName:='100 - Automaticky rezim - cakanie na start cyklu';
			SC_Valcovanie.IdleTime.PT:= T#500ms;
			SC_Valcovanie.AlarmTime.PT:= T#5s;
			Priznak_ValcovanieOK:= FALSE;

            SC_Valcovanie.IdleTime.IN:= NOT diValcovanie_PritomnostRotora;

			IF Valcovanie_KoniecCyklu THEN
				SC_Valcovanie.ResetStep:= TRUE;
				SC_Valcovanie.Step:= 0;
			ELSIF NOT VnutorneValcovanie_AKTIVNE THEN
				SC_Valcovanie.ResetStep:= TRUE;
				SC_Valcovanie.Step:= 120;
			ELSIF Stol_PoINIT AND NOT Valcovanie_UkoncilCyklus AND diValcovanie_PritomnostRotora AND diStol_SnimacPolohyStola THEN
				SC_Valcovanie.ResetStep:= TRUE;
				SC_Valcovanie.Step:= 101;
			ELSIF Stol_PoINIT AND NOT Valcovanie_UkoncilCyklus AND NOT diValcovanie_PritomnostRotora AND SC_Valcovanie.IdleTime.Q THEN
				SC_Valcovanie.ResetStep:= TRUE;
				SC_Valcovanie.Step:= 120;
			ELSIF Valcovanie_KoniecVyroby AND NOT Stol_Automat THEN
				SC_Valcovanie.ResetStep:= TRUE;
				SC_Valcovanie.Step:= 0;
			END_IF

		101:
			SC_Valcovanie.StepName:='101 - Automaticky rezim - zdvih rotora';
			SC_Valcovanie.IdleTime.PT:= T#500ms;
			SC_Valcovanie.AlarmTime.PT:= T#5s;

			IF NOT SC_Valcovanie.Switch1 THEN
				Rotor_ZDVIHNI:= TRUE;
				PocetCyklovValcovania:= PocetCyklovValcovania + 1;
				SC_Valcovanie.Switch1:= TRUE;
			END_IF

			IF diValcovanie_ZdvihHornaPoloha THEN
				SC_Valcovanie.ResetStep:= TRUE;
				SC_Valcovanie.Step:= 102;
			END_IF

		102:
			SC_Valcovanie.StepName:='102 - Automaticky rezim - zatvorenie gripra';
			SC_Valcovanie.IdleTime.PT:= T#500ms;
			SC_Valcovanie.AlarmTime.PT:= T#5s;

			IF NOT SC_Valcovanie.Switch1 THEN
				Zatvor_Griper:= TRUE;
				SC_Valcovanie.Switch1:= TRUE;
			END_IF

			IF diValcovanie_GriperZatvoreny THEN
				SC_Valcovanie.ResetStep:= TRUE;
				SC_Valcovanie.Step:= 103;
			END_IF

		103:
			SC_Valcovanie.StepName:='103 - Automaticky rezim - spustenie otacania nastroja, zostup do pozicie zaciatku valcovania, streknutie oleja';
			SC_Valcovanie.IdleTime.PT:= CasValcovania_ms;
			SC_Valcovanie.AlarmTime.PT:= T#5s;

			SC_Valcovanie.IdleTime.IN:= Valcovanie_ZdvihVPOZICI;
			Valcovanie_ZadanaPozMM:= TP_Valcovanie_PoziciaVnorenia; //50

			IF NOT SC_Valcovanie.Switch1 AND NOT diValcovanie_PritomnostNastroja AND SC_OvlServoZdvihu.Step = 1 THEN
				RotorOtacaj_VPRED:= TRUE;
				ServoZdvih_Polohuj:= TRUE;
				SC_Valcovanie.Switch1:= TRUE;
			END_IF

			IF PocetCyklovValcovania >= TP_Valcovanie_PocetCyklPredStrek THEN
				IF EDGEPOS (Valcovanie_AktualPozMM >= (TP_Valcovanie_PoziciaVnorenia - 50)) THEN
					doValcovanie_DavkaOleja:= TRUE;
					PocetCyklovValcovania:= 0;
				END_IF
			END_IF

			IF Valcovanie_ZdvihVPOZICI AND SC_Valcovanie.IdleTime.Q THEN
				Valcovanie_ZdvihVPOZICI:= FALSE;
				SC_Valcovanie.ResetStep:= TRUE;
				SC_Valcovanie.Step:= 107;
			END_IF

		107:
			SC_Valcovanie.StepName:='107 - Automaticky rezim - zdvih valcovacieho nastroja, otvorenie gripra, zasunutie zdvihu';
			SC_Valcovanie.IdleTime.PT:= T#500ms;
			SC_Valcovanie.AlarmTime.PT:= T#5s;
			SC_Valcovanie.IdleTime.IN:= TRUE;

			Valcovanie_ZadanaPozMM:= 15;

			IF NOT SC_Valcovanie.Switch1 AND SC_OvlServoZdvihu.Step = 1 THEN
				ServoZdvih_Polohuj:= TRUE;
				SC_Valcovanie.Switch1:= TRUE;
			END_IF

			IF EDGEPOS(Valcovanie_AktualPozMM < 60) THEN
				Otvor_Griper:= TRUE;
			END_IF

			IF EDGENEG(diValcovanie_GriperZatvoreny = TRUE) THEN
				Rotor_POLOZ:= TRUE;
			END_IF

			IF Valcovanie_ZdvihVPOZICI AND diValcovanie_GriperOtvoreny AND diValcovanie_ZdvihSpodnaPoloha THEN
				Valcovanie_ZdvihVPOZICI:= FALSE;
				SC_Valcovanie.ResetStep:= TRUE;
				SC_Valcovanie.Step:= 120;
			END_IF

		120:
			SC_Valcovanie.StepName:='120 - Automaticky rezim - vystavenie signalu ukoncenie pracovneho cyklu';
			SC_Valcovanie.IdleTime.PT:= T#500ms;
			SC_Valcovanie.AlarmTime.PT:= T#5s;

			IF Priznak_ValcovanieNG THEN
				Alarmy[77]:= TRUE;
				PoruchaStanicaValcovania:= TRUE;
			ELSE
				Valcovanie_UkoncilCyklus:= TRUE;
				SC_Valcovanie.ResetStep:= TRUE;
				SC_Valcovanie.Step:= 121;
			END_IF

		121:
			SC_Valcovanie.StepName:='121 - Automaticky rezim - cakanie na otocenie stola';
			SC_Valcovanie.IdleTime.PT:= T#500ms;
			SC_Valcovanie.AlarmTime.PT:= T#5s;

			IF diValcovanie_PritomnostNastroja THEN
				Alarmy[68]:= TRUE;
				PoruchaStanicaValcovania:= TRUE;
			END_IF

			IF NOT Valcovanie_UkoncilCyklus THEN
				SC_Valcovanie.ResetStep:= TRUE;
				SC_Valcovanie.Step:= 100;
			ELSIF Valcovanie_KoniecVyroby AND NOT Stol_Automat THEN
				SC_Valcovanie.ResetStep:= TRUE;
				SC_Valcovanie.Step:= 0;
			ELSIF Valcovanie_KoniecCyklu THEN
				SC_Valcovanie.ResetStep:= TRUE;
				SC_Valcovanie.Step:= 0;
			END_IF

			//********************************************************Ručný režim***********************************************************************************//
		700:
			SC_Valcovanie.StepName:='700 - Rucny rezim';

			//Ovládanie odstreku oleja//
			IF RR_StartOlejovania THEN
				doValcovanie_DavkaOleja:= TRUE;
				RR_StartOlejovania:= FALSE;
			END_IF

			//Polohovanie zdvihu valcovania//
			IF RR_PoziciaVychodzia AND SC_OvlServoZdvihu.Step = 1 THEN
				Valcovanie_Rychlost_MM_s:= TP_Valcovanie_RychlostZdvihu;
				Valcovanie_ZadanaPozMM:= 10;
				ServoZdvih_Polohuj:= TRUE;
			ELSIF RR_PoziciaValcovania AND SC_OvlServoZdvihu.Step = 1 THEN
				Valcovanie_Rychlost_MM_s:= TP_Valcovanie_RychlostZdvihu;
				Valcovanie_ZadanaPozMM:= TP_Valcovanie_PoziciaVnorenia;
				ServoZdvih_Polohuj:= TRUE;
			END_IF

	END_CASE

				END_PROGRAM

PROGRAM _EXIT
				(* Insert code here *)

				END_PROGRAM
```

#### Variables.var - Local variables
```iecst
VAR
	SC_OvlServoZdvihu : SequenceControlTyp;
	ServoZdvih_JoggDOLE : BOOL;
	ServoZdvih_JoggHORE : BOOL;
	ServoZdvih_Polohuj : BOOL;
	RR_PoziciaVychodzia : BOOL;
	RR_PoziciaValcovania : BOOL;
	SC_OvlZdvihu : SequenceControlTyp;
	Rotor_ZDVIHNI : BOOL;
	Rotor_POLOZ : BOOL;
	SC_OvlGripra : SequenceControlTyp;
	Otvor_Griper : BOOL;
	Zatvor_Griper : BOOL;
	SC_OvlOtacania : SequenceControlTyp;
	RotorOtacaj_VPRED : BOOL;
	RotorOtacaj_VZAD : BOOL;
	KonstantaZdvihu_MM : REAL;
	KonstantaZdvihu_Servo : REAL;
	CasStrekuOleja : TIME;
	PocetCyklovValcovania : UINT;
	RR_StartOlejovania : BOOL;
	CasStrikaniaOleja : TON;
	Priznak_ValcovanieNG : BOOL;
	Priznak_ValcovanieOK : BOOL;
END_VAR
```

#### OvladanieZdvihuServa.st
```iecst
ACTION OvladanieZdvihuServa:

	//Prepočet rýchlosti pojazdu manipulátora//
	KonstantaZdvihu_MM:= 10;  //10mm
	KonstantaZdvihu_Servo:= 1000; //počet jednotiek za 10mm

	Valcovanie_Rychlost_MM_s:= TP_Valcovanie_RychlostZdvihu;
	Valcovanie_ServoRychlostPolohov:= (Valcovanie_Rychlost_MM_s / KonstantaZdvihu_MM) * KonstantaZdvihu_Servo;
	Valcovanie_ServoRychlJoggingu:= (Valcovanie_RychlostJog_MM_s / KonstantaZdvihu_MM) * KonstantaZdvihu_Servo;
	Valcovanie_AktualPozMM;

	//Volanie funkcie SequenceControl//
	SequenceControl(SC:= SC_OvlServoZdvihu);

	CASE SC_OvlServoZdvihu.Step OF

		0:
			SC_OvlServoZdvihu.StepName:= '0 - Nulovanie';
			ServoZdvih_JoggDOLE:= FALSE;
			ServoZdvih_JoggHORE:= FALSE;
			ServoZdvih_Polohuj:= FALSE;
			Valcovanie_ZdvihHOME:= FALSE;
			Motion[3].cmd.home:= FALSE;
			Motion[3].cmd.moveAbsolute:= FALSE;
			Motion[3].cmd.moveJogNeg:= FALSE;
			Motion[3].cmd.moveJogPos:= FALSE;
			Valcovanie_PrebiehaHoming:= FALSE;
			IF NOT SC_OvlServoZdvihu.Switch1 AND Motion[3].status.DriveStatus.HomingOk THEN
				Motion[3].cmd.halt:= TRUE;
				SC_OvlServoZdvihu.Switch1:= TRUE;
			END_IF

			IF SC_Valcovanie.Step <> 0 THEN
				SC_OvlServoZdvihu.ResetStep:= TRUE;
				SC_OvlServoZdvihu.Step:= 1;
			END_IF

		1:
			SC_OvlServoZdvihu.StepName:= '1 - Rozhodnutie o cinnosti';
			IF ServoZdvih_JoggDOLE THEN
				SC_OvlServoZdvihu.Step:= 10;
			ELSIF ServoZdvih_JoggHORE THEN
				SC_OvlServoZdvihu.Step:= 20;
			ELSIF ServoZdvih_Polohuj THEN
				SC_OvlServoZdvihu.Step:= 30;
			ELSIF Valcovanie_ZdvihHOME THEN
				SC_OvlServoZdvihu.Step:= 40;
			END_IF

		10:
			SC_OvlServoZdvihu.StepName:= '10 - Jogging DOLE';
			SC_OvlServoZdvihu.IdleTime.PT:= T#3s;
			SC_OvlServoZdvihu.AlarmTime.PT:= T#3s;

			Motion[3].par.velocityJog:= Valcovanie_ServoRychlJoggingu;
			Motion[3].par.acc := (Valcovanie_ServoRychlJoggingu*10);
			Motion[3].par.dec := (Valcovanie_ServoRychlJoggingu*10);

			IF NOT SC_OvlServoZdvihu.Switch1 THEN
				Motion[3].cmd.moveJogPos:= TRUE;
				SC_OvlServoZdvihu.Switch1:= TRUE;
			END_IF

			IF NOT ServoZdvih_JoggDOLE OR diValcovanie_SpodnyLimitSnimac OR Valcovanie_AktualPozMM >= 200 THEN
				SC_OvlServoZdvihu.ResetStep:= TRUE;
				SC_OvlServoZdvihu.Step:= 0;
			END_IF

		20:
			SC_OvlServoZdvihu.StepName:= '20 - Jogging HORE';
			SC_OvlServoZdvihu.IdleTime.PT:= T#3s;
			SC_OvlServoZdvihu.AlarmTime.PT:= T#3s;

			Motion[3].par.velocityJog:= Valcovanie_ServoRychlJoggingu;
			Motion[3].par.acc := (Valcovanie_ServoRychlJoggingu*10);
			Motion[3].par.dec := (Valcovanie_ServoRychlJoggingu*10);

			IF NOT SC_OvlServoZdvihu.Switch1 THEN
				Motion[3].cmd.moveJogNeg:= TRUE;
				SC_OvlServoZdvihu.Switch1:= TRUE;
			END_IF

			IF NOT ServoZdvih_JoggHORE OR diValcovanie_HornyLimitSnimac OR Valcovanie_AktualPozMM < 5 THEN
				SC_OvlServoZdvihu.ResetStep:= TRUE;
				SC_OvlServoZdvihu.Step:= 0;
			END_IF

		30:
			SC_OvlServoZdvihu.StepName:= '30 - Start polohovanie zdvihu';
			SC_OvlServoZdvihu.IdleTime.PT:= T#3s;
			SC_OvlServoZdvihu.AlarmTime.PT:= T#3s;

			Motion[3].par.velocity:= Valcovanie_ServoRychlostPolohov;
			Motion[3].par.acc := (Valcovanie_ServoRychlostPolohov*20);
			Motion[3].par.dec := (Valcovanie_ServoRychlostPolohov*20);
			Motion[3].par.position:= (Valcovanie_ZadanaPozMM * 100);

			IF NOT SC_OvlServoZdvihu.Switch1 THEN
				Motion[3].cmd.moveAbsolute:= TRUE;
				SC_OvlServoZdvihu.Switch1:= TRUE;
			END_IF

			IF NOT Motion[3].state.StandStill THEN
				SC_OvlServoZdvihu.ResetStep:= TRUE;
				SC_OvlServoZdvihu.Step:= 31;
			ELSIF (Valcovanie_AktualPozMM = Valcovanie_ZadanaPozMM) THEN
				SC_OvlServoZdvihu.ResetStep:= TRUE;
				SC_OvlServoZdvihu.Step:= 31;
			END_IF

		31:

			SC_OvlServoZdvihu.StepName:= '31 - Ukoncenie polohovanie pojazdu';
			SC_OvlServoZdvihu.IdleTime.PT:= T#3s;
			SC_OvlServoZdvihu.AlarmTime.PT:= T#3s;

			IF Motion[3].status.ActTorque >= 5 THEN
				Motion[3].cmd.halt:= TRUE;
				Priznak_ValcovanieNG:= TRUE;
				SC_OvlServoZdvihu.ResetStep:= TRUE;
				SC_OvlServoZdvihu.Step:= 35;
			ELSIF Motion[3].state.StandStill AND (Valcovanie_AktualPozMM = Valcovanie_ZadanaPozMM) THEN
				Valcovanie_ZdvihVPOZICI:= TRUE;
				SC_OvlServoZdvihu.ResetStep:= TRUE;
				SC_OvlServoZdvihu.Step:= 0;
			END_IF

			IF diValcovanie_HornyLimitSnimac OR diValcovanie_SpodnyLimitSnimac THEN
				Alarmy[67]:= TRUE;
				PoruchaStanicaValcovania:= TRUE;
			END_IF

		35:
			SC_OvlServoZdvihu.StepName:= '35 - Cakanie na zastavenie serva po dosiahnuti limitneho momentu';
			SC_OvlServoZdvihu.IdleTime.PT:= T#1s;
			SC_OvlServoZdvihu.AlarmTime.PT:= T#3s;

			SC_OvlServoZdvihu.IdleTime.IN:= TRUE;

			IF SC_OvlServoZdvihu.IdleTime.Q AND Motion[3].state.StandStill THEN
				Motion[3].cmd.halt:= FALSE;
				Valcovanie_ZdvihVPOZICI:= TRUE;
				SC_OvlServoZdvihu.ResetStep:= TRUE;
				SC_OvlServoZdvihu.Step:= 0;
			END_IF

		40:
			SC_OvlServoZdvihu.StepName:= '40 - Start homingu';
			SC_OvlServoZdvihu.IdleTime.PT:= T#3s;
			SC_OvlServoZdvihu.AlarmTime.PT:= T#3s;

			IF NOT SC_OvlServoZdvihu.Switch1 THEN
				Motion[3].cmd.home:= TRUE;
				Valcovanie_PrebiehaHoming:= TRUE;
				SC_OvlServoZdvihu.Switch1:= TRUE;
			END_IF

			IF Motion[3].state.Homing THEN
				SC_OvlServoZdvihu.ResetStep:= TRUE;
				SC_OvlServoZdvihu.Step:= 41;
			END_IF

		41:
			SC_OvlServoZdvihu.StepName:= '41 - Ukoncenie homingu';
			SC_OvlServoZdvihu.IdleTime.PT:= T#3s;
			SC_OvlServoZdvihu.AlarmTime.PT:= T#3s;

			IF Motion[3].status.DriveStatus.HomingOk THEN
				SC_OvlServoZdvihu.ResetStep:= TRUE;
				SC_OvlServoZdvihu.Step:= 0;
			END_IF

	END_CASE

END_ACTION
```
